LIN {X 0,Y 250.853,Z 488.42,A -85,B 0,C 180,E1 -19750.986,E2 -19750.986} C_VEL
LIN {X 0,Y 251.245,Z 485.6,A -85,B 0,C 180,E1 -19751.504,E2 -19751.504} C_VEL
LIN {X 0,Y 250.177,Z 476.188,A -85,B 0,C 180,E1 -19753.375,E2 -19753.375} C_VEL
LIN {X 0,Y 248.189,Z 466.179,A -85,B 0,C 180,E1 -19755.22,E2 -19755.22} C_VEL
LIN {X 0,Y 245.226,Z 455.953,A -85,B 0,C 180,E1 -19757.02,E2 -19757.02} C_VEL
LIN {X 0,Y 240.964,Z 445.055,A -85,B 0,C 180,E1 -19758.907,E2 -19758.907} C_VEL
LIN {X 0,Y 237.476,Z 437.757,A -85,B 0,C 180,E1 -19760.172,E2 -19760.172} C_VEL
LIN {X 0,Y 236.049,Z 435.07,A -85,B 0,C 180,E1 -19760.656,E2 -19760.656} C_VEL
LIN {X 0,Y 235.755,Z 433.819,A -85,B 0,C 180,E1 -19760.811,E2 -19760.811} C_VEL
LIN {X 0,Y 235.735,Z 432.062,A -85,B 0,C 180,E1 -19763.605,E2 -19763.605} C_VEL
LIN {X 0,Y 235.472,Z 429.817,A -85,B 0,C 180,E1 -19767.505,E2 -19767.505} C_VEL
LIN {X 0,Y 235.182,Z 427.768,A -85,B 0,C 180,E1 -19771.437,E2 -19771.437} C_VEL
LIN {X 0,Y 235.056,Z 426.651,A -85,B 0,C 180,E1 -19773.762,E2 -19773.762} C_VEL
LIN {X 0,Y 234.975,Z 426.216,A -85,B 0,C 180,E1 -19775.246,E2 -19775.246} C_VEL
LIN {X 0,Y 234.995,Z 426.214,A -85,B 0,C 180,E1 -19778.969,E2 -19778.969} C_VEL
LIN {X 0,Y 235.093,Z 426.196,A -85,B 0,C 180,E1 -19783.06,E2 -19783.06} C_VEL
LIN {X 0,Y 235.142,Z 426.195,A -85,B 0,C 180,E1 -19787.924,E2 -19787.924} C_VEL
LIN {X 0,Y 235.374,Z 426.166,A -85,B 0,C 180,E1 -19791.414,E2 -19791.414} C_VEL
LIN {X 0,Y 235.401,Z 426.162,A -85,B 0,C 180,E1 -19793.142,E2 -19793.142} C_VEL
LIN {X 0,Y 235.593,Z 426.139,A -85,B 0,C 180,E1 -19798.291,E2 -19798.291} C_VEL
LIN {X 0,Y 235.593,Z 426.14,A -85,B 0,C 180,E1 -19801.71,E2 -19801.71} C_VEL
LIN {X 0,Y 235.4,Z 426.156,A -85,B 0,C 180,E1 -19806.859,E2 -19806.859} C_VEL
LIN {X 0,Y 235.236,Z 426.183,A -85,B 0,C 180,E1 -19810.327,E2 -19810.327} C_VEL
LIN {X 0,Y 235.112,Z 426.199,A -85,B 0,C 180,E1 -19815.607,E2 -19815.607} C_VEL
LIN {X 0,Y 235.007,Z 426.214,A -85,B 0,C 180,E1 -19819.206,E2 -19819.206} C_VEL
LIN {X 0,Y 234.959,Z 426.222,A -85,B 0,C 180,E1 -19822.883,E2 -19822.883} C_VEL
LIN {X 0,Y 234.969,Z 426.219,A -85,B 0,C 180,E1 -19826.658,E2 -19826.658} C_VEL
LIN {X 0,Y 234.992,Z 426.424,A -85,B 0,C 180,E1 -19829.853,E2 -19829.853} C_VEL
LIN {X 0,Y 235.419,Z 429.003,A -85,B 0,C 180,E1 -19834.556,E2 -19834.556} C_VEL
LIN {X 0,Y 235.897,Z 431.588,A -85,B 0,C 180,E1 -19838.73,E2 -19838.73} C_VEL
LIN {X 0,Y 236.352,Z 434.709,A -85,B 0,C 180,E1 -19843.151,E2 -19843.151} C_VEL
LIN {X 0,Y 236.828,Z 437.629,A -85,B 0,C 180,E1 -19846.958,E2 -19846.958} C_VEL
LIN {X 0,Y 237.155,Z 440.504,A -85,B 0,C 180,E1 -19850.399,E2 -19850.399} C_VEL
LIN {X 0,Y 237.192,Z 441.841,A -85,B 0,C 180,E1 -19851.906,E2 -19851.906} C_VEL
LIN {X 0,Y 237.306,Z 443.408,A -85,B 0,C 180,E1 -19852.73,E2 -19852.73} C_VEL
LIN {X 0,Y 237.585,Z 446.002,A -85,B 0,C 180,E1 -19853.4,E2 -19853.4} C_VEL
LIN {X 0,Y 238.041,Z 450.995,A -85,B 0,C 180,E1 -19854.165,E2 -19854.165} C_VEL
LIN {X 0,Y 238.686,Z 465.72,A -85,B 0,C 180,E1 -19855.664,E2 -19855.664} C_VEL
LIN {X 0,Y 239.11,Z 468.433,A -85,B 0,C 180,E1 -19856.063,E2 -19856.063} C_VEL
LIN {X 0,Y 241.3,Z 479.581,A -85,B 0,C 180,E1 -19857.932,E2 -19857.932} C_VEL
LIN {X 0,Y 242.552,Z 490.657,A -85,B 0,C 180,E1 -19859.937,E2 -19859.937} C_VEL
LIN {X 0,Y 242.646,Z 501.177,A -85,B 0,C 180,E1 -19862.009,E2 -19862.009} C_VEL
LIN {X 0,Y 242.306,Z 505.014,A -85,B 0,C 180,E1 -19862.818,E2 -19862.818} C_VEL
LIN {X 0,Y 239.128,Z 514.446,A -85,B 0,C 180,E1 -19864.776,E2 -19864.776} C_VEL
LIN {X 0,Y 235.867,Z 523.545,A -85,B 0,C 180,E1 -19867.21,E2 -19867.21} C_VEL
LIN {X 0,Y 233.14,Z 530.894,A -85,B 0,C 180,E1 -19869.716,E2 -19869.716} C_VEL
LIN {X 0,Y 230.801,Z 536.822,A -85,B 0,C 180,E1 -19872.272,E2 -19872.272} C_VEL
LIN {X 0,Y 228.794,Z 541.531,A -85,B 0,C 180,E1 -19874.865,E2 -19874.865} C_VEL
LIN {X 0,Y 227.42,Z 545.155,A -85,B 0,C 180,E1 -19877.507,E2 -19877.507} C_VEL
LIN {X 0,Y 226.704,Z 547.044,A -85,B 0,C 180,E1 -19879.28,E2 -19879.28} C_VEL
LIN {X 0,Y 225.834,Z 549.522,A -85,B 0,C 180,E1 -19882.849,E2 -19882.849} C_VEL
LIN {X 0,Y 225.597,Z 550.455,A -85,B 0,C 180,E1 -19886.428,E2 -19886.428} C_VEL
LIN {X 0,Y 225.664,Z 550.323,A -85,B 0,C 180,E1 -19888.215,E2 -19888.215} C_VEL
LIN {X 0,Y 225.758,Z 549.776,A -85,B 0,C 180,E1 -19890,E2 -19890} C_VEL
LIN {X 0,Y 225.69,Z 548.83,A -85,B 0,C 180,E1 -19891.784,E2 -19891.784} C_VEL
LIN {X 0,Y 225.67,Z 546.343,A -85,B 0,C 180,E1 -19894.743,E2 -19894.743} C_VEL
LIN {X 0,Y 225.956,Z 542.13,A -85,B 0,C 180,E1 -19898.045,E2 -19898.045} C_VEL
LIN {X 0,Y 226.522,Z 537.447,A -85,B 0,C 180,E1 -19900.728,E2 -19900.728} C_VEL
LIN {X 0,Y 227.568,Z 530.357,A -85,B 0,C 180,E1 -19903.847,E2 -19903.847} C_VEL
LIN {X 0,Y 229.062,Z 522.678,A -85,B 0,C 180,E1 -19906.487,E2 -19906.487} C_VEL
LIN {X 0,Y 230.612,Z 514.353,A -85,B 0,C 180,E1 -19908.773,E2 -19908.773} C_VEL
LIN {X 0,Y 232.453,Z 504.046,A -85,B 0,C 180,E1 -19911.04,E2 -19911.04} C_VEL
LIN {X 0,Y 233.96,Z 494.379,A -85,B 0,C 180,E1 -19912.752,E2 -19912.752} C_VEL
LIN {X 0,Y 233.445,Z 483.574,A -85,B 0,C 180,E1 -19914.452,E2 -19914.452} C_VEL
LIN {X 0,Y 232.439,Z 471.5,A -85,B 0,C 180,E1 -19915.995,E2 -19915.995} C_VEL
LIN {X 0,Y 230.575,Z 458.277,A -85,B 0,C 180,E1 -19917.362,E2 -19917.362} C_VEL
LIN {X 0,Y 227.792,Z 445.678,A -85,B 0,C 180,E1 -19918.423,E2 -19918.423} C_VEL
LIN {X 0,Y 227.578,Z 444.108,A -85,B 0,C 180,E1 -19918.517,E2 -19918.517} C_VEL
LIN {X 0,Y 228.74,Z 438.72,A -85,B 0,C 180,E1 -19923.575,E2 -19923.575} C_VEL
LIN {X 0,Y 229.126,Z 436.565,A -85,B 0,C 180,E1 -19925.646,E2 -19925.646} C_VEL
LIN {X 0,Y 229.232,Z 434.369,A -85,B 0,C 180,E1 -19927.818,E2 -19927.818} C_VEL
LIN {X 0,Y 228.704,Z 431.101,A -85,B 0,C 180,E1 -19931.273,E2 -19931.273} C_VEL
LIN {X 0,Y 227.914,Z 427.097,A -85,B 0,C 180,E1 -19935.8,E2 -19935.8} C_VEL
LIN {X 0,Y 227.851,Z 427.105,A -85,B 0,C 180,E1 -19940.452,E2 -19940.452} C_VEL
LIN {X 0,Y 227.877,Z 427.099,A -85,B 0,C 180,E1 -19944.127,E2 -19944.127} C_VEL
LIN {X 0,Y 227.867,Z 427.1,A -85,B 0,C 180,E1 -19948.377,E2 -19948.377} C_VEL
LIN {X 0,Y 227.881,Z 427.085,A -85,B 0,C 180,E1 -19952.444,E2 -19952.444} C_VEL
LIN {X 0,Y 227.91,Z 427.094,A -85,B 0,C 180,E1 -19956.367,E2 -19956.367} C_VEL
LIN {X 0,Y 227.936,Z 427.088,A -85,B 0,C 180,E1 -19960.174,E2 -19960.174} C_VEL
LIN {X 0,Y 228.04,Z 427.056,A -85,B 0,C 180,E1 -19963.896,E2 -19963.896} C_VEL
LIN {X 0,Y 228.162,Z 427.062,A -85,B 0,C 180,E1 -19969.349,E2 -19969.349} C_VEL
LIN {X 0,Y 228.354,Z 427.033,A -85,B 0,C 180,E1 -19972.928,E2 -19972.928} C_VEL
LIN {X 0,Y 228.55,Z 426.996,A -85,B 0,C 180,E1 -19978.238,E2 -19978.238} C_VEL
LIN {X 0,Y 228.55,Z 427.011,A -85,B 0,C 180,E1 -19981.762,E2 -19981.762} C_VEL
LIN {X 0,Y 228.35,Z 427.034,A -85,B 0,C 180,E1 -19987.071,E2 -19987.071} C_VEL
LIN {X 0,Y 228.154,Z 427.04,A -85,B 0,C 180,E1 -19990.651,E2 -19990.651} C_VEL
LIN {X 0,Y 228.057,Z 427.067,A -85,B 0,C 180,E1 -19994.272,E2 -19994.272} C_VEL
LIN {X 0,Y 227.998,Z 427.085,A -85,B 0,C 180,E1 -19997.953,E2 -19997.953} C_VEL
LIN {X 0,Y 227.925,Z 427.09,A -85,B 0,C 180,E1 -20002.329,E2 -20002.329} C_VEL
LIN {X 0,Y 227.937,Z 427.09,A -85,B 0,C 180,E1 -20006.603,E2 -20006.603} C_VEL
LIN {X 0,Y 227.893,Z 427.096,A -85,B 0,C 180,E1 -20010.292,E2 -20010.292} C_VEL
LIN {X 0,Y 227.886,Z 427.098,A -85,B 0,C 180,E1 -20013.719,E2 -20013.719} C_VEL
LIN {X 0,Y 227.868,Z 427.1,A -85,B 0,C 180,E1 -20018.086,E2 -20018.086} C_VEL
LIN {X 0,Y 227.93,Z 427.091,A -85,B 0,C 180,E1 -20022.714,E2 -20022.714} C_VEL
LIN {X 0,Y 227.931,Z 427.093,A -85,B 0,C 180,E1 -20027.287,E2 -20027.287} C_VEL
LIN {X 0,Y 227.869,Z 427.1,A -85,B 0,C 180,E1 -20031.915,E2 -20031.915} C_VEL
LIN {X 0,Y 227.888,Z 427.096,A -85,B 0,C 180,E1 -20036.374,E2 -20036.374} C_VEL
LIN {X 0,Y 227.917,Z 427.094,A -85,B 0,C 180,E1 -20040.439,E2 -20040.439} C_VEL
LIN {X 0,Y 227.923,Z 427.093,A -85,B 0,C 180,E1 -20044.426,E2 -20044.426} C_VEL
LIN {X 0,Y 228.038,Z 427.237,A -85,B 0,C 180,E1 -20048.296,E2 -20048.296} C_VEL
LIN {X 0,Y 227.441,Z 431.627,A -85,B 0,C 180,E1 -20053.854,E2 -20053.854} C_VEL
LIN {X 0,Y 227.218,Z 432.967,A -85,B 0,C 180,E1 -20055.503,E2 -20055.503} C_VEL
LIN {X 0,Y 231.479,Z 448.755,A -85,B 0,C 180,E1 -20057.006,E2 -20057.006} C_VEL
LIN {X 0,Y 233.767,Z 459.789,A -85,B 0,C 180,E1 -20058.272,E2 -20058.272} C_VEL
LIN {X 0,Y 235.175,Z 470.256,A -85,B 0,C 180,E1 -20059.671,E2 -20059.671} C_VEL
LIN {X 0,Y 235.635,Z 476.071,A -85,B 0,C 180,E1 -20060.55,E2 -20060.55} C_VEL
LIN {X 0,Y 233.896,Z 487.249,A -85,B 0,C 180,E1 -20062.335,E2 -20062.335} C_VEL
LIN {X 0,Y 232.04,Z 497.341,A -85,B 0,C 180,E1 -20064.351,E2 -20064.351} C_VEL
LIN {X 0,Y 230.343,Z 506,A -85,B 0,C 180,E1 -20066.502,E2 -20066.502} C_VEL
LIN {X 0,Y 228.668,Z 514.397,A -85,B 0,C 180,E1 -20069.12,E2 -20069.12} C_VEL
LIN {X 0,Y 227.487,Z 521.146,A -85,B 0,C 180,E1 -20071.771,E2 -20071.771} C_VEL
LIN {X 0,Y 226.632,Z 526.542,A -85,B 0,C 180,E1 -20074.447,E2 -20074.447} C_VEL
LIN {X 0,Y 226.023,Z 530.762,A -85,B 0,C 180,E1 -20077.145,E2 -20077.145} C_VEL
LIN {X 0,Y 225.696,Z 533.003,A -85,B 0,C 180,E1 -20078.957,E2 -20078.957} C_VEL
LIN {X 0,Y 225.457,Z 534.751,A -85,B 0,C 180,E1 -20080.78,E2 -20080.78} C_VEL
LIN {X 0,Y 225.393,Z 536.082,A -85,B 0,C 180,E1 -20082.607,E2 -20082.607} C_VEL
LIN {X 0,Y 225.404,Z 537.155,A -85,B 0,C 180,E1 -20084.858,E2 -20084.858} C_VEL
LIN {X 0,Y 225.646,Z 537.574,A -85,B 0,C 180,E1 -20088.147,E2 -20088.147} C_VEL
LIN {X 0,Y 226.379,Z 536.717,A -85,B 0,C 180,E1 -20091.353,E2 -20091.353} C_VEL
LIN {X 0,Y 227.101,Z 535.261,A -85,B 0,C 180,E1 -20093.722,E2 -20093.722} C_VEL
LIN {X 0,Y 228.657,Z 532.057,A -85,B 0,C 180,E1 -20096.958,E2 -20096.958} C_VEL
LIN {X 0,Y 230.763,Z 527.351,A -85,B 0,C 180,E1 -20100.166,E2 -20100.166} C_VEL
LIN {X 0,Y 233.107,Z 521.927,A -85,B 0,C 180,E1 -20102.866,E2 -20102.866} C_VEL
LIN {X 0,Y 235.838,Z 515.039,A -85,B 0,C 180,E1 -20105.528,E2 -20105.528} C_VEL
LIN {X 0,Y 238.67,Z 507.605,A -85,B 0,C 180,E1 -20107.787,E2 -20107.787} C_VEL
LIN {X 0,Y 241.524,Z 499.363,A -85,B 0,C 180,E1 -20109.804,E2 -20109.804} C_VEL
LIN {X 0,Y 244.42,Z 490.134,A -85,B 0,C 180,E1 -20111.618,E2 -20111.618} C_VEL
LIN {X 0,Y 244.886,Z 487.509,A -85,B 0,C 180,E1 -20112.103,E2 -20112.103} C_VEL
LIN {X 0,Y 244.042,Z 478.755,A -85,B 0,C 180,E1 -20113.949,E2 -20113.949} C_VEL
LIN {X 0,Y 242.279,Z 468.964,A -85,B 0,C 180,E1 -20115.878,E2 -20115.878} C_VEL
LIN {X 0,Y 239.09,Z 457.518,A -85,B 0,C 180,E1 -20118.031,E2 -20118.031} C_VEL
LIN {X 0,Y 234.687,Z 446.24,A -85,B 0,C 180,E1 -20120.133,E2 -20120.133} C_VEL
LIN {X 0,Y 232.428,Z 441.672,A -85,B 0,C 180,E1 -20121.021,E2 -20121.021} C_VEL
LIN {X 0,Y 230.777,Z 438.365,A -85,B 0,C 180,E1 -20121.648,E2 -20121.648} C_VEL
LIN {X 0,Y 229.134,Z 435.533,A -85,B 0,C 180,E1 -20122.231,E2 -20122.231} C_VEL
LIN {X 0,Y 228.744,Z 434.032,A -85,B 0,C 180,E1 -20122.505,E2 -20122.505} C_VEL
LIN {X 0,Y 228.598,Z 431.802,A -85,B 0,C 180,E1 -20126.4,E2 -20126.4} C_VEL
LIN {X 0,Y 228.31,Z 429.669,A -85,B 0,C 180,E1 -20130.494,E2 -20130.494} C_VEL
LIN {X 0,Y 228.049,Z 427.829,A -85,B 0,C 180,E1 -20134.441,E2 -20134.441} C_VEL
LIN {X 0,Y 227.904,Z 427.095,A -85,B 0,C 180,E1 -20136.367,E2 -20136.367} C_VEL
LIN {X 0,Y 227.934,Z 427.089,A -85,B 0,C 180,E1 -20140.174,E2 -20140.174} C_VEL
LIN {X 0,Y 228.051,Z 427.076,A -85,B 0,C 180,E1 -20143.898,E2 -20143.898} C_VEL
LIN {X 0,Y 228.16,Z 427.058,A -85,B 0,C 180,E1 -20149.35,E2 -20149.35} C_VEL
LIN {X 0,Y 228.352,Z 427.041,A -85,B 0,C 180,E1 -20152.929,E2 -20152.929} C_VEL
LIN {X 0,Y 228.551,Z 427.017,A -85,B 0,C 180,E1 -20158.238,E2 -20158.238} C_VEL
LIN {X 0,Y 228.552,Z 427.017,A -85,B 0,C 180,E1 -20161.762,E2 -20161.762} C_VEL
LIN {X 0,Y 228.351,Z 427.033,A -85,B 0,C 180,E1 -20167.072,E2 -20167.072} C_VEL
LIN {X 0,Y 228.161,Z 427.064,A -85,B 0,C 180,E1 -20170.651,E2 -20170.651} C_VEL
LIN {X 0,Y 228.063,Z 427.077,A -85,B 0,C 180,E1 -20174.273,E2 -20174.273} C_VEL
LIN {X 0,Y 228.001,Z 427.088,A -85,B 0,C 180,E1 -20177.954,E2 -20177.954} C_VEL
LIN {X 0,Y 227.928,Z 427.096,A -85,B 0,C 180,E1 -20182.33,E2 -20182.33} C_VEL
LIN {X 0,Y 227.942,Z 427.094,A -85,B 0,C 180,E1 -20186.603,E2 -20186.603} C_VEL
LIN {X 0,Y 227.885,Z 427.102,A -85,B 0,C 180,E1 -20187.556,E2 -20187.556} C_VEL
LIN {X 0,Y 228.128,Z 428.34,A -85,B 0,C 180,E1 -20190.391,E2 -20190.391} C_VEL
LIN {X 0,Y 228.419,Z 430.171,A -85,B 0,C 180,E1 -20193.827,E2 -20193.827} C_VEL
LIN {X 0,Y 228.828,Z 432.576,A -85,B 0,C 180,E1 -20197.899,E2 -20197.899} C_VEL
LIN {X 0,Y 229.332,Z 435.555,A -85,B 0,C 180,E1 -20202.393,E2 -20202.393} C_VEL
LIN {X 0,Y 229.662,Z 437.646,A -85,B 0,C 180,E1 -20205.265,E2 -20205.265} C_VEL
LIN {X 0,Y 229.943,Z 439.568,A -85,B 0,C 180,E1 -20207.747,E2 -20207.747} C_VEL
LIN {X 0,Y 230.216,Z 442.935,A -85,B 0,C 180,E1 -20211.803,E2 -20211.803} C_VEL
LIN {X 0,Y 230.232,Z 443.288,A -85,B 0,C 180,E1 -20211.988,E2 -20211.988} C_VEL
LIN {X 0,Y 231.387,Z 446.527,A -85,B 0,C 180,E1 -20212.454,E2 -20212.454} C_VEL
LIN {X 0,Y 232.603,Z 448.763,A -85,B 0,C 180,E1 -20212.877,E2 -20212.877} C_VEL
LIN {X 0,Y 236.801,Z 459.979,A -85,B 0,C 180,E1 -20214.704,E2 -20214.704} C_VEL
LIN {X 0,Y 239.11,Z 468.433,A -85,B 0,C 180,E1 -20216.063,E2 -20216.063} C_VEL
LIN {X 0,Y 239.668,Z 473.57,A -85,B 0,C 180,E1 -20216.801,E2 -20216.801} C_VEL
LIN {X 0,Y 238.465,Z 482.57,A -85,B 0,C 180,E1 -20217.875,E2 -20217.875} C_VEL
LIN {X 0,Y 236.768,Z 491.002,A -85,B 0,C 180,E1 -20219.037,E2 -20219.037} C_VEL
LIN {X 0,Y 236.424,Z 495.65,A -85,B 0,C 180,E1 -20219.888,E2 -20219.888} C_VEL
LIN {X 0,Y 235.983,Z 505.59,A -85,B 0,C 180,E1 -20222.027,E2 -20222.027} C_VEL
LIN {X 0,Y 232.755,Z 514.85,A -85,B 0,C 180,E1 -20224.035,E2 -20224.035} C_VEL
LIN {X 0,Y 229.35,Z 523.832,A -85,B 0,C 180,E1 -20226.524,E2 -20226.524} C_VEL
LIN {X 0,Y 226.495,Z 531.095,A -85,B 0,C 180,E1 -20229.094,E2 -20229.094} C_VEL
LIN {X 0,Y 224.042,Z 536.946,A -85,B 0,C 180,E1 -20231.718,E2 -20231.718} C_VEL
LIN {X 0,Y 221.927,Z 541.586,A -85,B 0,C 180,E1 -20234.385,E2 -20234.385} C_VEL
LIN {X 0,Y 220.463,Z 545.144,A -85,B 0,C 180,E1 -20237.106,E2 -20237.106} C_VEL
LIN {X 0,Y 219.709,Z 546.986,A -85,B 0,C 180,E1 -20238.935,E2 -20238.935} C_VEL
LIN {X 0,Y 218.79,Z 549.388,A -85,B 0,C 180,E1 -20242.618,E2 -20242.618} C_VEL
LIN {X 0,Y 218.5,Z 550.258,A -85,B 0,C 180,E1 -20246.311,E2 -20246.311} C_VEL
LIN {X 0,Y 218.579,Z 550.076,A -85,B 0,C 180,E1 -20248.157,E2 -20248.157} C_VEL
LIN {X 0,Y 218.67,Z 549.502,A -85,B 0,C 180,E1 -20250,E2 -20250} C_VEL
LIN {X 0,Y 218.605,Z 548.528,A -85,B 0,C 180,E1 -20251.842,E2 -20251.842} C_VEL
LIN {X 0,Y 218.576,Z 546.262,A -85,B 0,C 180,E1 -20254.609,E2 -20254.609} C_VEL
LIN {X 0,Y 218.78,Z 542.993,A -85,B 0,C 180,E1 -20257.382,E2 -20257.382} C_VEL
LIN {X 0,Y 219.273,Z 538.633,A -85,B 0,C 180,E1 -20260.153,E2 -20260.153} C_VEL
LIN {X 0,Y 220.05,Z 533.053,A -85,B 0,C 180,E1 -20262.918,E2 -20262.918} C_VEL
LIN {X 0,Y 221.421,Z 526.086,A -85,B 0,C 180,E1 -20265.651,E2 -20265.651} C_VEL
LIN {X 0,Y 222.863,Z 518.953,A -85,B 0,C 180,E1 -20267.906,E2 -20267.906} C_VEL
LIN {X 0,Y 224.43,Z 510.287,A -85,B 0,C 180,E1 -20270.148,E2 -20270.148} C_VEL
LIN {X 0,Y 226.435,Z 499.599,A -85,B 0,C 180,E1 -20272.346,E2 -20272.346} C_VEL
LIN {X 0,Y 227.069,Z 494.531,A -85,B 0,C 180,E1 -20273.242,E2 -20273.242} C_VEL
LIN {X 0,Y 226.539,Z 483.294,A -85,B 0,C 180,E1 -20275.074,E2 -20275.074} C_VEL
LIN {X 0,Y 225.552,Z 471.16,A -85,B 0,C 180,E1 -20276.675,E2 -20276.675} C_VEL
LIN {X 0,Y 223.737,Z 458.469,A -85,B 0,C 180,E1 -20278.045,E2 -20278.045} C_VEL
LIN {X 0,Y 220.857,Z 445.431,A -85,B 0,C 180,E1 -20279.199,E2 -20279.199} C_VEL
LIN {X 0,Y 220.63,Z 443.898,A -85,B 0,C 180,E1 -20279.322,E2 -20279.322} C_VEL
LIN {X 0,Y 221.425,Z 440.452,A -85,B 0,C 180,E1 -20282.654,E2 -20282.654} C_VEL
LIN {X 0,Y 222.079,Z 437.223,A -85,B 0,C 180,E1 -20285.834,E2 -20285.834} C_VEL
LIN {X 0,Y 222.202,Z 435.346,A -85,B 0,C 180,E1 -20287.746,E2 -20287.746} C_VEL
LIN {X 0,Y 221.597,Z 431.693,A -85,B 0,C 180,E1 -20291.759,E2 -20291.759} C_VEL
LIN {X 0,Y 220.881,Z 427.973,A -85,B 0,C 180,E1 -20296.196,E2 -20296.196} C_VEL
LIN {X 0,Y 220.805,Z 427.983,A -85,B 0,C 180,E1 -20300.462,E2 -20300.462} C_VEL
LIN {X 0,Y 220.798,Z 427.984,A -85,B 0,C 180,E1 -20305.044,E2 -20305.044} C_VEL
LIN {X 0,Y 220.865,Z 427.969,A -85,B 0,C 180,E1 -20309.394,E2 -20309.394} C_VEL
LIN {X 0,Y 220.891,Z 427.96,A -85,B 0,C 180,E1 -20313.549,E2 -20313.549} C_VEL
LIN {X 0,Y 220.874,Z 427.97,A -85,B 0,C 180,E1 -20317.553,E2 -20317.553} C_VEL
LIN {X 0,Y 220.976,Z 427.938,A -85,B 0,C 180,E1 -20322.574,E2 -20322.574} C_VEL
LIN {X 0,Y 221.003,Z 427.952,A -85,B 0,C 180,E1 -20327.138,E2 -20327.138} C_VEL
LIN {X 0,Y 221.253,Z 427.923,A -85,B 0,C 180,E1 -20330.861,E2 -20330.861} C_VEL
LIN {X 0,Y 221.307,Z 427.911,A -85,B 0,C 180,E1 -20332.702,E2 -20332.702} C_VEL
LIN {X 0,Y 221.508,Z 427.871,A -85,B 0,C 180,E1 -20338.181,E2 -20338.181} C_VEL
LIN {X 0,Y 221.508,Z 427.889,A -85,B 0,C 180,E1 -20341.818,E2 -20341.818} C_VEL
LIN {X 0,Y 221.301,Z 427.912,A -85,B 0,C 180,E1 -20347.298,E2 -20347.298} C_VEL
LIN {X 0,Y 221.101,Z 427.916,A -85,B 0,C 180,E1 -20350.994,E2 -20350.994} C_VEL
LIN {X 0,Y 221.011,Z 427.953,A -85,B 0,C 180,E1 -20356.63,E2 -20356.63} C_VEL
LIN {X 0,Y 220.887,Z 427.966,A -85,B 0,C 180,E1 -20360.486,E2 -20360.486} C_VEL
LIN {X 0,Y 220.862,Z 427.973,A -85,B 0,C 180,E1 -20364.435,E2 -20364.435} C_VEL
LIN {X 0,Y 220.823,Z 427.971,A -85,B 0,C 180,E1 -20368.515,E2 -20368.515} C_VEL
LIN {X 0,Y 220.819,Z 427.977,A -85,B 0,C 180,E1 -20372.755,E2 -20372.755} C_VEL
LIN {X 0,Y 220.834,Z 427.974,A -85,B 0,C 180,E1 -20377.288,E2 -20377.288} C_VEL
LIN {X 0,Y 220.87,Z 427.972,A -85,B 0,C 180,E1 -20381.929,E2 -20381.929} C_VEL
LIN {X 0,Y 220.872,Z 427.973,A -85,B 0,C 180,E1 -20385.573,E2 -20385.573} C_VEL
LIN {X 0,Y 220.858,Z 427.974,A -85,B 0,C 180,E1 -20389.792,E2 -20389.792} C_VEL
LIN {X 0,Y 220.832,Z 427.976,A -85,B 0,C 180,E1 -20392.796,E2 -20392.796} C_VEL
LIN {X 0,Y 220.822,Z 427.979,A -85,B 0,C 180,E1 -20397.246,E2 -20397.246} C_VEL
LIN {X 0,Y 220.835,Z 427.978,A -85,B 0,C 180,E1 -20401.487,E2 -20401.487} C_VEL
LIN {X 0,Y 220.865,Z 427.975,A -85,B 0,C 180,E1 -20405.566,E2 -20405.566} C_VEL
LIN {X 0,Y 220.968,Z 428.041,A -85,B 0,C 180,E1 -20408.056,E2 -20408.056} C_VEL
LIN {X 0,Y 220.428,Z 432.056,A -85,B 0,C 180,E1 -20413.325,E2 -20413.325} C_VEL
LIN {X 0,Y 220.284,Z 433.239,A -85,B 0,C 180,E1 -20414.77,E2 -20414.77} C_VEL
LIN {X 0,Y 223.877,Z 446.278,A -85,B 0,C 180,E1 -20416.004,E2 -20416.004} C_VEL
LIN {X 0,Y 226.646,Z 458.785,A -85,B 0,C 180,E1 -20417.464,E2 -20417.464} C_VEL
LIN {X 0,Y 228.186,Z 469.686,A -85,B 0,C 180,E1 -20418.954,E2 -20418.954} C_VEL
LIN {X 0,Y 228.781,Z 477.32,A -85,B 0,C 180,E1 -20420.151,E2 -20420.151} C_VEL
LIN {X 0,Y 226.956,Z 488.347,A -85,B 0,C 180,E1 -20421.989,E2 -20421.989} C_VEL
LIN {X 0,Y 224.962,Z 498.737,A -85,B 0,C 180,E1 -20424.173,E2 -20424.173} C_VEL
LIN {X 0,Y 223.232,Z 507.152,A -85,B 0,C 180,E1 -20426.39,E2 -20426.39} C_VEL
LIN {X 0,Y 221.521,Z 515.38,A -85,B 0,C 180,E1 -20429.091,E2 -20429.091} C_VEL
LIN {X 0,Y 220.343,Z 521.989,A -85,B 0,C 180,E1 -20431.828,E2 -20431.828} C_VEL
LIN {X 0,Y 219.503,Z 527.258,A -85,B 0,C 180,E1 -20434.591,E2 -20434.591} C_VEL
LIN {X 0,Y 218.866,Z 531.366,A -85,B 0,C 180,E1 -20437.38,E2 -20437.38} C_VEL
LIN {X 0,Y 218.537,Z 533.5,A -85,B 0,C 180,E1 -20439.253,E2 -20439.253} C_VEL
LIN {X 0,Y 218.328,Z 535.192,A -85,B 0,C 180,E1 -20441.136,E2 -20441.136} C_VEL
LIN {X 0,Y 218.274,Z 536.473,A -85,B 0,C 180,E1 -20443.026,E2 -20443.026} C_VEL
LIN {X 0,Y 218.32,Z 537.358,A -85,B 0,C 180,E1 -20445.042,E2 -20445.042} C_VEL
LIN {X 0,Y 218.636,Z 537.758,A -85,B 0,C 180,E1 -20448.75,E2 -20448.75} C_VEL
LIN {X 0,Y 219.372,Z 536.945,A -85,B 0,C 180,E1 -20451.71,E2 -20451.71} C_VEL
LIN {X 0,Y 220.305,Z 535.236,A -85,B 0,C 180,E1 -20454.501,E2 -20454.501} C_VEL
LIN {X 0,Y 221.799,Z 532.335,A -85,B 0,C 180,E1 -20457.475,E2 -20457.475} C_VEL
LIN {X 0,Y 223.595,Z 528.59,A -85,B 0,C 180,E1 -20460.192,E2 -20460.192} C_VEL
LIN {X 0,Y 226.21,Z 522.951,A -85,B 0,C 180,E1 -20463.24,E2 -20463.24} C_VEL
LIN {X 0,Y 229.282,Z 515.724,A -85,B 0,C 180,E1 -20466.161,E2 -20466.161} C_VEL
LIN {X 0,Y 232.646,Z 507.256,A -85,B 0,C 180,E1 -20468.798,E2 -20468.798} C_VEL
LIN {X 0,Y 235.882,Z 498.375,A -85,B 0,C 180,E1 -20470.956,E2 -20470.956} C_VEL
LIN {X 0,Y 238.545,Z 489.774,A -85,B 0,C 180,E1 -20472.658,E2 -20472.658} C_VEL
LIN {X 0,Y 238.001,Z 481.816,A -85,B 0,C 180,E1 -20474.443,E2 -20474.443} C_VEL
LIN {X 0,Y 236.481,Z 472.206,A -85,B 0,C 180,E1 -20476.472,E2 -20476.472} C_VEL
LIN {X 0,Y 233.805,Z 461.655,A -85,B 0,C 180,E1 -20478.601,E2 -20478.601} C_VEL
LIN {X 0,Y 230.13,Z 451.192,A -85,B 0,C 180,E1 -20480.678,E2 -20480.678} C_VEL
LIN {X 0,Y 226.052,Z 442.859,A -85,B 0,C 180,E1 -20482.443,E2 -20482.443} C_VEL
LIN {X 0,Y 223.94,Z 438.84,A -85,B 0,C 180,E1 -20483.299,E2 -20483.299} C_VEL
LIN {X 0,Y 222.162,Z 435.944,A -85,B 0,C 180,E1 -20483.971,E2 -20483.971} C_VEL
LIN {X 0,Y 221.734,Z 434.343,A -85,B 0,C 180,E1 -20484.241,E2 -20484.241} C_VEL
LIN {X 0,Y 221.428,Z 431.852,A -85,B 0,C 180,E1 -20488.976,E2 -20488.976} C_VEL
LIN {X 0,Y 221.184,Z 429.682,A -85,B 0,C 180,E1 -20493.587,E2 -20493.587} C_VEL
LIN {X 0,Y 220.904,Z 428.075,A -85,B 0,C 180,E1 -20497.556,E2 -20497.556} C_VEL
LIN {X 0,Y 220.981,Z 427.955,A -85,B 0,C 180,E1 -20502.572,E2 -20502.572} C_VEL
LIN {X 0,Y 221.021,Z 427.953,A -85,B 0,C 180,E1 -20507.139,E2 -20507.139} C_VEL
LIN {X 0,Y 221.234,Z 427.929,A -85,B 0,C 180,E1 -20510.861,E2 -20510.861} C_VEL
LIN {X 0,Y 221.287,Z 427.922,A -85,B 0,C 180,E1 -20512.702,E2 -20512.702} C_VEL
LIN {X 0,Y 221.51,Z 427.894,A -85,B 0,C 180,E1 -20518.182,E2 -20518.182} C_VEL
LIN {X 0,Y 221.51,Z 427.894,A -85,B 0,C 180,E1 -20521.818,E2 -20521.818} C_VEL
LIN {X 0,Y 221.286,Z 427.912,A -85,B 0,C 180,E1 -20527.299,E2 -20527.299} C_VEL
LIN {X 0,Y 221.11,Z 427.944,A -85,B 0,C 180,E1 -20530.995,E2 -20530.995} C_VEL
LIN {X 0,Y 221.015,Z 427.958,A -85,B 0,C 180,E1 -20536.63,E2 -20536.63} C_VEL
LIN {X 0,Y 220.891,Z 427.973,A -85,B 0,C 180,E1 -20540.487,E2 -20540.487} C_VEL
LIN {X 0,Y 220.866,Z 427.977,A -85,B 0,C 180,E1 -20544.435,E2 -20544.435} C_VEL
LIN {X 0,Y 220.934,Z 428.431,A -85,B 0,C 180,E1 -20547.041,E2 -20547.041} C_VEL
LIN {X 0,Y 221.218,Z 430.234,A -85,B 0,C 180,E1 -20550.933,E2 -20550.933} C_VEL
LIN {X 0,Y 221.569,Z 432.301,A -85,B 0,C 180,E1 -20554.817,E2 -20554.817} C_VEL
LIN {X 0,Y 221.879,Z 433.935,A -85,B 0,C 180,E1 -20557.64,E2 -20557.64} C_VEL
LIN {X 0,Y 222.256,Z 436.44,A -85,B 0,C 180,E1 -20561.61,E2 -20561.61} C_VEL
LIN {X 0,Y 222.791,Z 439.913,A -85,B 0,C 180,E1 -20566.514,E2 -20566.514} C_VEL
LIN {X 0,Y 223.151,Z 442.815,A -85,B 0,C 180,E1 -20570.21,E2 -20570.21} C_VEL
LIN {X 0,Y 224.201,Z 445.876,A -85,B 0,C 180,E1 -20570.682,E2 -20570.682} C_VEL
LIN {X 0,Y 225.802,Z 448.582,A -85,B 0,C 180,E1 -20571.267,E2 -20571.267} C_VEL
LIN {X 0,Y 228.196,Z 454.18,A -85,B 0,C 180,E1 -20572.291,E2 -20572.291} C_VEL
LIN {X 0,Y 231.577,Z 463.952,A -85,B 0,C 180,E1 -20574.026,E2 -20574.026} C_VEL
LIN {X 0,Y 234.295,Z 475.596,A -85,B 0,C 180,E1 -20576.056,E2 -20576.056} C_VEL
LIN {X 0,Y 235.858,Z 486.753,A -85,B 0,C 180,E1 -20578.107,E2 -20578.107} C_VEL
LIN {X 0,Y 236.424,Z 495.65,A -85,B 0,C 180,E1 -20579.888,E2 -20579.888} C_VEL
LIN {X 0,Y 236.097,Z 498.733,A -85,B 0,C 180,E1 -20580.474,E2 -20580.474} C_VEL
LIN {X 0,Y 234.381,Z 503.411,A -85,B 0,C 180,E1 -20581.257,E2 -20581.257} C_VEL
LIN {X 0,Y 231.792,Z 507.929,A -85,B 0,C 180,E1 -20581.98,E2 -20581.98} C_VEL
LIN {X 0,Y 226.978,Z 515.185,A -85,B 0,C 180,E1 -20583.307,E2 -20583.307} C_VEL
LIN {X 0,Y 224.82,Z 519.243,A -85,B 0,C 180,E1 -20584.314,E2 -20584.314} C_VEL
LIN {X 0,Y 221.482,Z 527.49,A -85,B 0,C 180,E1 -20586.959,E2 -20586.959} C_VEL
LIN {X 0,Y 218.942,Z 533.341,A -85,B 0,C 180,E1 -20589.323,E2 -20589.323} C_VEL
LIN {X 0,Y 216.491,Z 538.691,A -85,B 0,C 180,E1 -20592.037,E2 -20592.037} C_VEL
LIN {X 0,Y 214.457,Z 542.891,A -85,B 0,C 180,E1 -20594.801,E2 -20594.801} C_VEL
LIN {X 0,Y 213.525,Z 545.133,A -85,B 0,C 180,E1 -20596.679,E2 -20596.679} C_VEL
LIN {X 0,Y 212.732,Z 546.914,A -85,B 0,C 180,E1 -20598.567,E2 -20598.567} C_VEL
LIN {X 0,Y 211.721,Z 549.256,A -85,B 0,C 180,E1 -20602.37,E2 -20602.37} C_VEL
LIN {X 0,Y 211.421,Z 550.032,A -85,B 0,C 180,E1 -20605.759,E2 -20605.759} C_VEL
LIN {X 0,Y 211.476,Z 549.827,A -85,B 0,C 180,E1 -20608.095,E2 -20608.095} C_VEL
LIN {X 0,Y 211.585,Z 549.224,A -85,B 0,C 180,E1 -20610,E2 -20610} C_VEL
LIN {X 0,Y 211.501,Z 548.22,A -85,B 0,C 180,E1 -20611.904,E2 -20611.904} C_VEL
LIN {X 0,Y 211.474,Z 546.206,A -85,B 0,C 180,E1 -20614.432,E2 -20614.432} C_VEL
LIN {X 0,Y 211.705,Z 542.559,A -85,B 0,C 180,E1 -20617.63,E2 -20617.63} C_VEL
LIN {X 0,Y 212.241,Z 538.131,A -85,B 0,C 180,E1 -20620.493,E2 -20620.493} C_VEL
LIN {X 0,Y 213.085,Z 532.476,A -85,B 0,C 180,E1 -20623.348,E2 -20623.348} C_VEL
LIN {X 0,Y 214.561,Z 525.404,A -85,B 0,C 180,E1 -20626.165,E2 -20626.165} C_VEL
LIN {X 0,Y 216.101,Z 518.172,A -85,B 0,C 180,E1 -20628.486,E2 -20628.486} C_VEL
LIN {X 0,Y 217.492,Z 510.5,A -85,B 0,C 180,E1 -20630.534,E2 -20630.534} C_VEL
LIN {X 0,Y 219.608,Z 499.715,A -85,B 0,C 180,E1 -20632.831,E2 -20632.831} C_VEL
LIN {X 0,Y 220.165,Z 494.66,A -85,B 0,C 180,E1 -20633.765,E2 -20633.765} C_VEL
LIN {X 0,Y 219.744,Z 484.299,A -85,B 0,C 180,E1 -20635.53,E2 -20635.53} C_VEL
LIN {X 0,Y 218.848,Z 472.055,A -85,B 0,C 180,E1 -20637.246,E2 -20637.246} C_VEL
LIN {X 0,Y 217.045,Z 459.375,A -85,B 0,C 180,E1 -20638.699,E2 -20638.699} C_VEL
LIN {X 0,Y 214.261,Z 446.394,A -85,B 0,C 180,E1 -20639.916,E2 -20639.916} C_VEL
LIN {X 0,Y 213.709,Z 443.696,A -85,B 0,C 180,E1 -20640.167,E2 -20640.167} C_VEL
LIN {X 0,Y 214.567,Z 440.038,A -85,B 0,C 180,E1 -20643.835,E2 -20643.835} C_VEL
LIN {X 0,Y 215.127,Z 436.798,A -85,B 0,C 180,E1 -20647.17,E2 -20647.17} C_VEL
LIN {X 0,Y 214.688,Z 433.472,A -85,B 0,C 180,E1 -20650.897,E2 -20650.897} C_VEL
LIN {X 0,Y 214.038,Z 429.921,A -85,B 0,C 180,E1 -20655.094,E2 -20655.094} C_VEL
LIN {X 0,Y 213.819,Z 428.854,A -85,B 0,C 180,E1 -20656.674,E2 -20656.674} C_VEL
LIN {X 0,Y 213.728,Z 428.863,A -85,B 0,C 180,E1 -20662.108,E2 -20662.108} C_VEL
LIN {X 0,Y 213.754,Z 428.858,A -85,B 0,C 180,E1 -20666.017,E2 -20666.017} C_VEL
LIN {X 0,Y 213.777,Z 428.849,A -85,B 0,C 180,E1 -20670.453,E2 -20670.453} C_VEL
LIN {X 0,Y 213.798,Z 428.846,A -85,B 0,C 180,E1 -20674.701,E2 -20674.701} C_VEL
LIN {X 0,Y 213.808,Z 428.85,A -85,B 0,C 180,E1 -20678.803,E2 -20678.803} C_VEL
LIN {X 0,Y 213.934,Z 428.812,A -85,B 0,C 180,E1 -20682.802,E2 -20682.802} C_VEL
LIN {X 0,Y 213.943,Z 428.828,A -85,B 0,C 180,E1 -20686.706,E2 -20686.706} C_VEL
LIN {X 0,Y 214.192,Z 428.805,A -85,B 0,C 180,E1 -20690.557,E2 -20690.557} C_VEL
LIN {X 0,Y 214.243,Z 428.793,A -85,B 0,C 180,E1 -20692.46,E2 -20692.46} C_VEL
LIN {X 0,Y 214.441,Z 428.75,A -85,B 0,C 180,E1 -20698.122,E2 -20698.122} C_VEL
LIN {X 0,Y 214.549,Z 428.748,A -85,B 0,C 180,E1 -20700,E2 -20700} C_VEL
LIN {X 0,Y 214.441,Z 428.769,A -85,B 0,C 180,E1 -20701.878,E2 -20701.878} C_VEL
LIN {X 0,Y 214.235,Z 428.792,A -85,B 0,C 180,E1 -20707.54,E2 -20707.54} C_VEL
LIN {X 0,Y 214.018,Z 428.796,A -85,B 0,C 180,E1 -20711.363,E2 -20711.363} C_VEL
LIN {X 0,Y 213.927,Z 428.829,A -85,B 0,C 180,E1 -20715.237,E2 -20715.237} C_VEL
LIN {X 0,Y 213.835,Z 428.847,A -85,B 0,C 180,E1 -20719.187,E2 -20719.187} C_VEL
LIN {X 0,Y 213.843,Z 428.843,A -85,B 0,C 180,E1 -20723.227,E2 -20723.227} C_VEL
LIN {X 0,Y 213.825,Z 428.849,A -85,B 0,C 180,E1 -20727.45,E2 -20727.45} C_VEL
LIN {X 0,Y 213.766,Z 428.858,A -85,B 0,C 180,E1 -20731.738,E2 -20731.738} C_VEL
LIN {X 0,Y 213.751,Z 428.855,A -85,B 0,C 180,E1 -20736.287,E2 -20736.287} C_VEL
LIN {X 0,Y 213.821,Z 428.849,A -85,B 0,C 180,E1 -20741.099,E2 -20741.099} C_VEL
LIN {X 0,Y 213.833,Z 428.849,A -85,B 0,C 180,E1 -20743.693,E2 -20743.693} C_VEL
LIN {X 0,Y 213.838,Z 428.846,A -85,B 0,C 180,E1 -20746.357,E2 -20746.357} C_VEL
LIN {X 0,Y 213.821,Z 428.85,A -85,B 0,C 180,E1 -20749.11,E2 -20749.11} C_VEL
LIN {X 0,Y 213.752,Z 428.858,A -85,B 0,C 180,E1 -20753.715,E2 -20753.715} C_VEL
LIN {X 0,Y 213.794,Z 428.853,A -85,B 0,C 180,E1 -20758.725,E2 -20758.725} C_VEL
LIN {X 0,Y 213.824,Z 428.85,A -85,B 0,C 180,E1 -20762.604,E2 -20762.604} C_VEL
LIN {X 0,Y 213.938,Z 429.021,A -85,B 0,C 180,E1 -20768.058,E2 -20768.058} C_VEL
LIN {X 0,Y 213.348,Z 433.225,A -85,B 0,C 180,E1 -20773.74,E2 -20773.74} C_VEL
LIN {X 0,Y 213.328,Z 433.365,A -85,B 0,C 180,E1 -20773.923,E2 -20773.923} C_VEL
LIN {X 0,Y 217.107,Z 446.939,A -85,B 0,C 180,E1 -20775.289,E2 -20775.289} C_VEL
LIN {X 0,Y 219.788,Z 459.09,A -85,B 0,C 180,E1 -20776.772,E2 -20776.772} C_VEL
LIN {X 0,Y 221.351,Z 469.972,A -85,B 0,C 180,E1 -20778.323,E2 -20778.323} C_VEL
LIN {X 0,Y 222.003,Z 478.185,A -85,B 0,C 180,E1 -20779.669,E2 -20779.669} C_VEL
LIN {X 0,Y 220.21,Z 488.428,A -85,B 0,C 180,E1 -20781.431,E2 -20781.431} C_VEL
LIN {X 0,Y 218.26,Z 498.231,A -85,B 0,C 180,E1 -20783.529,E2 -20783.529} C_VEL
LIN {X 0,Y 216.442,Z 506.79,A -85,B 0,C 180,E1 -20785.811,E2 -20785.811} C_VEL
LIN {X 0,Y 214.654,Z 515.112,A -85,B 0,C 180,E1 -20788.593,E2 -20788.593} C_VEL
LIN {X 0,Y 213.391,Z 521.807,A -85,B 0,C 180,E1 -20791.416,E2 -20791.416} C_VEL
LIN {X 0,Y 212.353,Z 527.937,A -85,B 0,C 180,E1 -20794.746,E2 -20794.746} C_VEL
LIN {X 0,Y 211.709,Z 531.93,A -85,B 0,C 180,E1 -20797.631,E2 -20797.631} C_VEL
LIN {X 0,Y 211.403,Z 533.989,A -85,B 0,C 180,E1 -20799.568,E2 -20799.568} C_VEL
LIN {X 0,Y 211.199,Z 535.631,A -85,B 0,C 180,E1 -20801.517,E2 -20801.517} C_VEL
LIN {X 0,Y 211.169,Z 536.85,A -85,B 0,C 180,E1 -20803.472,E2 -20803.472} C_VEL
LIN {X 0,Y 211.234,Z 537.613,A -85,B 0,C 180,E1 -20805.436,E2 -20805.436} C_VEL
LIN {X 0,Y 211.376,Z 537.977,A -85,B 0,C 180,E1 -20807.412,E2 -20807.412} C_VEL
LIN {X 0,Y 211.656,Z 537.943,A -85,B 0,C 180,E1 -20809.393,E2 -20809.393} C_VEL
LIN {X 0,Y 212.369,Z 537.174,A -85,B 0,C 180,E1 -20812.088,E2 -20812.088} C_VEL
LIN {X 0,Y 213.537,Z 535.211,A -85,B 0,C 180,E1 -20815.332,E2 -20815.332} C_VEL
LIN {X 0,Y 215,Z 532.586,A -85,B 0,C 180,E1 -20818.045,E2 -20818.045} C_VEL
LIN {X 0,Y 217.149,Z 528.335,A -85,B 0,C 180,E1 -20821.187,E2 -20821.187} C_VEL
LIN {X 0,Y 219.819,Z 522.89,A -85,B 0,C 180,E1 -20824.142,E2 -20824.142} C_VEL
LIN {X 0,Y 222.73,Z 516.413,A -85,B 0,C 180,E1 -20826.835,E2 -20826.835} C_VEL
LIN {X 0,Y 226.155,Z 508.313,A -85,B 0,C 180,E1 -20829.457,E2 -20829.457} C_VEL
LIN {X 0,Y 229.618,Z 499.341,A -85,B 0,C 180,E1 -20831.736,E2 -20831.736} C_VEL
LIN {X 0,Y 232.23,Z 491.21,A -85,B 0,C 180,E1 -20833.422,E2 -20833.422} C_VEL
LIN {X 0,Y 231.735,Z 483.303,A -85,B 0,C 180,E1 -20835.299,E2 -20835.299} C_VEL
LIN {X 0,Y 230.469,Z 474.47,A -85,B 0,C 180,E1 -20837.274,E2 -20837.274} C_VEL
LIN {X 0,Y 228.179,Z 464.783,A -85,B 0,C 180,E1 -20839.367,E2 -20839.367} C_VEL
LIN {X 0,Y 225.12,Z 455.435,A -85,B 0,C 180,E1 -20841.364,E2 -20841.364} C_VEL
LIN {X 0,Y 221.21,Z 447.013,A -85,B 0,C 180,E1 -20843.296,E2 -20843.296} C_VEL
LIN {X 0,Y 219.445,Z 443.603,A -85,B 0,C 180,E1 -20844.093,E2 -20844.093} C_VEL
LIN {X 0,Y 217.257,Z 439.512,A -85,B 0,C 180,E1 -20845.058,E2 -20845.058} C_VEL
LIN {X 0,Y 215.303,Z 436.747,A -85,B 0,C 180,E1 -20845.835,E2 -20845.835} C_VEL
LIN {X 0,Y 214.614,Z 434.647,A -85,B 0,C 180,E1 -20846.243,E2 -20846.243} C_VEL
LIN {X 0,Y 214.369,Z 432.54,A -85,B 0,C 180,E1 -20850.543,E2 -20850.543} C_VEL
LIN {X 0,Y 214.117,Z 430.714,A -85,B 0,C 180,E1 -20854.742,E2 -20854.742} C_VEL
LIN {X 0,Y 213.866,Z 429.179,A -85,B 0,C 180,E1 -20858.809,E2 -20858.809} C_VEL
LIN {X 0,Y 213.94,Z 428.831,A -85,B 0,C 180,E1 -20862.804,E2 -20862.804} C_VEL
LIN {X 0,Y 213.957,Z 428.83,A -85,B 0,C 180,E1 -20866.707,E2 -20866.707} C_VEL
LIN {X 0,Y 214.165,Z 428.808,A -85,B 0,C 180,E1 -20870.557,E2 -20870.557} C_VEL
LIN {X 0,Y 214.225,Z 428.802,A -85,B 0,C 180,E1 -20872.46,E2 -20872.46} C_VEL
LIN {X 0,Y 214.443,Z 428.775,A -85,B 0,C 180,E1 -20878.122,E2 -20878.122} C_VEL
LIN {X 0,Y 214.547,Z 428.761,A -85,B 0,C 180,E1 -20880,E2 -20880} C_VEL
LIN {X 0,Y 214.444,Z 428.774,A -85,B 0,C 180,E1 -20881.878,E2 -20881.878} C_VEL
LIN {X 0,Y 214.224,Z 428.791,A -85,B 0,C 180,E1 -20887.541,E2 -20887.541} C_VEL
LIN {X 0,Y 214.043,Z 428.824,A -85,B 0,C 180,E1 -20891.362,E2 -20891.362} C_VEL
LIN {X 0,Y 213.932,Z 428.838,A -85,B 0,C 180,E1 -20895.237,E2 -20895.237} C_VEL
LIN {X 0,Y 213.838,Z 428.851,A -85,B 0,C 180,E1 -20899.188,E2 -20899.188} C_VEL
LIN {X 0,Y 213.846,Z 428.852,A -85,B 0,C 180,E1 -20903.228,E2 -20903.228} C_VEL
LIN {X 0,Y 214.066,Z 430.316,A -85,B 0,C 180,E1 -20907.573,E2 -20907.573} C_VEL
LIN {X 0,Y 214.326,Z 432.189,A -85,B 0,C 180,E1 -20911.646,E2 -20911.646} C_VEL
LIN {X 0,Y 214.749,Z 434.54,A -85,B 0,C 180,E1 -20916.092,E2 -20916.092} C_VEL
LIN {X 0,Y 215.227,Z 437.325,A -85,B 0,C 180,E1 -20920.775,E2 -20920.775} C_VEL
LIN {X 0,Y 215.734,Z 440.706,A -85,B 0,C 180,E1 -20925.783,E2 -20925.783} C_VEL
LIN {X 0,Y 216.024,Z 442.653,A -85,B 0,C 180,E1 -20928.267,E2 -20928.267} C_VEL
LIN {X 0,Y 217.182,Z 445.761,A -85,B 0,C 180,E1 -20928.81,E2 -20928.81} C_VEL
LIN {X 0,Y 218.866,Z 448.223,A -85,B 0,C 180,E1 -20929.457,E2 -20929.457} C_VEL
LIN {X 0,Y 220.848,Z 452.341,A -85,B 0,C 180,E1 -20930.329,E2 -20930.329} C_VEL
LIN {X 0,Y 223.752,Z 459.429,A -85,B 0,C 180,E1 -20931.744,E2 -20931.744} C_VEL
LIN {X 0,Y 226.775,Z 469.735,A -85,B 0,C 180,E1 -20933.685,E2 -20933.685} C_VEL
LIN {X 0,Y 228.746,Z 480.031,A -85,B 0,C 180,E1 -20935.629,E2 -20935.629} C_VEL
LIN {X 0,Y 229.93,Z 491.069,A -85,B 0,C 180,E1 -20937.834,E2 -20937.834} C_VEL
LIN {X 0,Y 230.064,Z 499.826,A -85,B 0,C 180,E1 -20939.722,E2 -20939.722} C_VEL
LIN {X 0,Y 229.655,Z 506.171,A -85,B 0,C 180,E1 -20941.185,E2 -20941.185} C_VEL
LIN {X 0,Y 227.081,Z 513.577,A -85,B 0,C 180,E1 -20942.839,E2 -20942.839} C_VEL
LIN {X 0,Y 224.82,Z 519.243,A -85,B 0,C 180,E1 -20944.314,E2 -20944.314} C_VEL
LIN {X 0,Y 222.714,Z 523.035,A -85,B 0,C 180,E1 -20945.362,E2 -20945.362} C_VEL
LIN {X 0,Y 217.73,Z 528.783,A -85,B 0,C 180,E1 -20947.03,E2 -20947.03} C_VEL
LIN {X 0,Y 212.825,Z 533.844,A -85,B 0,C 180,E1 -20948.875,E2 -20948.875} C_VEL
LIN {X 0,Y 210.882,Z 536.556,A -85,B 0,C 180,E1 -20950.18,E2 -20950.18} C_VEL
LIN {X 0,Y 208.255,Z 541.671,A -85,B 0,C 180,E1 -20953.331,E2 -20953.331} C_VEL
LIN {X 0,Y 206.584,Z 545.112,A -85,B 0,C 180,E1 -20956.223,E2 -20956.223} C_VEL
LIN {X 0,Y 205.114,Z 548.175,A -85,B 0,C 180,E1 -20960.135,E2 -20960.135} C_VEL
LIN {X 0,Y 204.408,Z 549.687,A -85,B 0,C 180,E1 -20964.079,E2 -20964.079} C_VEL
LIN {X 0,Y 204.337,Z 549.827,A -85,B 0,C 180,E1 -20966.055,E2 -20966.055} C_VEL
LIN {X 0,Y 204.377,Z 549.579,A -85,B 0,C 180,E1 -20968.029,E2 -20968.029} C_VEL
LIN {X 0,Y 204.501,Z 548.947,A -85,B 0,C 180,E1 -20970,E2 -20970} C_VEL
LIN {X 0,Y 204.401,Z 547.912,A -85,B 0,C 180,E1 -20971.97,E2 -20971.97} C_VEL
LIN {X 0,Y 204.38,Z 546.129,A -85,B 0,C 180,E1 -20974.265,E2 -20974.265} C_VEL
LIN {X 0,Y 204.652,Z 542.126,A -85,B 0,C 180,E1 -20977.895,E2 -20977.895} C_VEL
LIN {X 0,Y 205.214,Z 537.628,A -85,B 0,C 180,E1 -20980.856,E2 -20980.856} C_VEL
LIN {X 0,Y 206.381,Z 530.783,A -85,B 0,C 180,E1 -20984.293,E2 -20984.293} C_VEL
LIN {X 0,Y 207.964,Z 523.327,A -85,B 0,C 180,E1 -20987.199,E2 -20987.199} C_VEL
LIN {X 0,Y 209.626,Z 515.715,A -85,B 0,C 180,E1 -20989.588,E2 -20989.588} C_VEL
LIN {X 0,Y 211.044,Z 508.437,A -85,B 0,C 180,E1 -20991.488,E2 -20991.488} C_VEL
LIN {X 0,Y 213.006,Z 498.641,A -85,B 0,C 180,E1 -20993.581,E2 -20993.581} C_VEL
LIN {X 0,Y 213.296,Z 493.443,A -85,B 0,C 180,E1 -20994.581,E2 -20994.581} C_VEL
LIN {X 0,Y 212.847,Z 482.41,A -85,B 0,C 180,E1 -20996.483,E2 -20996.483} C_VEL
LIN {X 0,Y 211.8,Z 470.069,A -85,B 0,C 180,E1 -20998.218,E2 -20998.218} C_VEL
LIN {X 0,Y 210.003,Z 457.999,A -85,B 0,C 180,E1 -20999.628,E2 -20999.628} C_VEL
LIN {X 0,Y 206.971,Z 444.713,A -85,B 0,C 180,E1 -21000.922,E2 -21000.922} C_VEL
LIN {X 0,Y 206.829,Z 443.473,A -85,B 0,C 180,E1 -21001.075,E2 -21001.075} C_VEL
LIN {X 0,Y 207.786,Z 439.622,A -85,B 0,C 180,E1 -21005.098,E2 -21005.098} C_VEL
LIN {X 0,Y 208.073,Z 437.454,A -85,B 0,C 180,E1 -21007.442,E2 -21007.442} C_VEL
LIN {X 0,Y 207.81,Z 435.248,A -85,B 0,C 180,E1 -21009.982,E2 -21009.982} C_VEL
LIN {X 0,Y 207.101,Z 431.479,A -85,B 0,C 180,E1 -21014.55,E2 -21014.55} C_VEL
LIN {X 0,Y 206.76,Z 429.733,A -85,B 0,C 180,E1 -21016.851,E2 -21016.851} C_VEL
LIN {X 0,Y 206.677,Z 429.742,A -85,B 0,C 180,E1 -21022.259,E2 -21022.259} C_VEL
LIN {X 0,Y 206.696,Z 429.74,A -85,B 0,C 180,E1 -21027.041,E2 -21027.041} C_VEL
LIN {X 0,Y 206.763,Z 429.713,A -85,B 0,C 180,E1 -21032.096,E2 -21032.096} C_VEL
LIN {X 0,Y 206.782,Z 429.726,A -85,B 0,C 180,E1 -21036.583,E2 -21036.583} C_VEL
LIN {X 0,Y 206.865,Z 429.697,A -85,B 0,C 180,E1 -21042.195,E2 -21042.195} C_VEL
LIN {X 0,Y 206.884,Z 429.704,A -85,B 0,C 180,E1 -21046.243,E2 -21046.243} C_VEL
LIN {X 0,Y 207.128,Z 429.685,A -85,B 0,C 180,E1 -21050.232,E2 -21050.232} C_VEL
LIN {X 0,Y 207.184,Z 429.674,A -85,B 0,C 180,E1 -21052.201,E2 -21052.201} C_VEL
LIN {X 0,Y 207.378,Z 429.628,A -85,B 0,C 180,E1 -21058.058,E2 -21058.058} C_VEL
LIN {X 0,Y 207.514,Z 429.624,A -85,B 0,C 180,E1 -21060,E2 -21060} C_VEL
LIN {X 0,Y 207.083,Z 429.69,A -85,B 0,C 180,E1 -21063.892,E2 -21063.892} C_VEL
LIN {X 0,Y 207.173,Z 429.669,A -85,B 0,C 180,E1 -21067.798,E2 -21067.798} C_VEL
LIN {X 0,Y 206.938,Z 429.677,A -85,B 0,C 180,E1 -21071.757,E2 -21071.757} C_VEL
LIN {X 0,Y 206.861,Z 429.711,A -85,B 0,C 180,E1 -21075.771,E2 -21075.771} C_VEL
LIN {X 0,Y 206.779,Z 429.728,A -85,B 0,C 180,E1 -21079.869,E2 -21079.869} C_VEL
LIN {X 0,Y 206.759,Z 429.73,A -85,B 0,C 180,E1 -21084.072,E2 -21084.072} C_VEL
LIN {X 0,Y 206.732,Z 429.726,A -85,B 0,C 180,E1 -21088.42,E2 -21088.42} C_VEL
LIN {X 0,Y 206.702,Z 429.736,A -85,B 0,C 180,E1 -21092.957,E2 -21092.957} C_VEL
LIN {X 0,Y 206.722,Z 429.734,A -85,B 0,C 180,E1 -21097.73,E2 -21097.73} C_VEL
LIN {X 0,Y 206.746,Z 429.732,A -85,B 0,C 180,E1 -21101.597,E2 -21101.597} C_VEL
LIN {X 0,Y 206.743,Z 429.732,A -85,B 0,C 180,E1 -21105.55,E2 -21105.55} C_VEL
LIN {X 0,Y 206.741,Z 429.733,A -85,B 0,C 180,E1 -21109.769,E2 -21109.769} C_VEL
LIN {X 0,Y 206.729,Z 429.732,A -85,B 0,C 180,E1 -21114.696,E2 -21114.696} C_VEL
LIN {X 0,Y 206.722,Z 429.735,A -85,B 0,C 180,E1 -21119.34,E2 -21119.34} C_VEL
LIN {X 0,Y 206.731,Z 429.734,A -85,B 0,C 180,E1 -21123.773,E2 -21123.773} C_VEL
LIN {X 0,Y 206.842,Z 429.733,A -85,B 0,C 180,E1 -21127.628,E2 -21127.628} C_VEL
LIN {X 0,Y 206.401,Z 433.366,A -85,B 0,C 180,E1 -21132.734,E2 -21132.734} C_VEL
LIN {X 0,Y 206.4,Z 433.828,A -85,B 0,C 180,E1 -21133.058,E2 -21133.058} C_VEL
LIN {X 0,Y 210.123,Z 446.878,A -85,B 0,C 180,E1 -21134.439,E2 -21134.439} C_VEL
LIN {X 0,Y 212.912,Z 459.099,A -85,B 0,C 180,E1 -21136.001,E2 -21136.001} C_VEL
LIN {X 0,Y 214.572,Z 470.635,A -85,B 0,C 180,E1 -21137.709,E2 -21137.709} C_VEL
LIN {X 0,Y 215.217,Z 478.894,A -85,B 0,C 180,E1 -21139.127,E2 -21139.127} C_VEL
LIN {X 0,Y 213.104,Z 490.369,A -85,B 0,C 180,E1 -21141.202,E2 -21141.202} C_VEL
LIN {X 0,Y 211.19,Z 499.577,A -85,B 0,C 180,E1 -21143.312,E2 -21143.312} C_VEL
LIN {X 0,Y 209.338,Z 507.921,A -85,B 0,C 180,E1 -21145.668,E2 -21145.668} C_VEL
LIN {X 0,Y 207.507,Z 516.088,A -85,B 0,C 180,E1 -21148.545,E2 -21148.545} C_VEL
LIN {X 0,Y 206.448,Z 521.626,A -85,B 0,C 180,E1 -21150.976,E2 -21150.976} C_VEL
LIN {X 0,Y 205.446,Z 527.051,A -85,B 0,C 180,E1 -21153.923,E2 -21153.923} C_VEL
LIN {X 0,Y 204.75,Z 531.296,A -85,B 0,C 180,E1 -21156.899,E2 -21156.899} C_VEL
LIN {X 0,Y 204.247,Z 534.481,A -85,B 0,C 180,E1 -21159.907,E2 -21159.907} C_VEL
LIN {X 0,Y 204.086,Z 536.068,A -85,B 0,C 180,E1 -21161.924,E2 -21161.924} C_VEL
LIN {X 0,Y 204.137,Z 537.759,A -85,B 0,C 180,E1 -21165.426,E2 -21165.426} C_VEL
LIN {X 0,Y 204.36,Z 538.214,A -85,B 0,C 180,E1 -21168.03,E2 -21168.03} C_VEL
LIN {X 0,Y 204.722,Z 538.109,A -85,B 0,C 180,E1 -21170.078,E2 -21170.078} C_VEL
LIN {X 0,Y 205.387,Z 537.4,A -85,B 0,C 180,E1 -21172.498,E2 -21172.498} C_VEL
LIN {X 0,Y 206.814,Z 535.185,A -85,B 0,C 180,E1 -21176.217,E2 -21176.217} C_VEL
LIN {X 0,Y 208.198,Z 532.859,A -85,B 0,C 180,E1 -21178.639,E2 -21178.639} C_VEL
LIN {X 0,Y 210.798,Z 528.077,A -85,B 0,C 180,E1 -21182.238,E2 -21182.238} C_VEL
LIN {X 0,Y 214.057,Z 521.643,A -85,B 0,C 180,E1 -21185.645,E2 -21185.645} C_VEL
LIN {X 0,Y 217.345,Z 514.695,A -85,B 0,C 180,E1 -21188.435,E2 -21188.435} C_VEL
LIN {X 0,Y 220.538,Z 507.259,A -85,B 0,C 180,E1 -21190.789,E2 -21190.789} C_VEL
LIN {X 0,Y 224.48,Z 497.323,A -85,B 0,C 180,E1 -21193.224,E2 -21193.224} C_VEL
LIN {X 0,Y 225.906,Z 493.325,A -85,B 0,C 180,E1 -21194.05,E2 -21194.05} C_VEL
LIN {X 0,Y 225.589,Z 485.41,A -85,B 0,C 180,E1 -21196.052,E2 -21196.052} C_VEL
LIN {X 0,Y 224.379,Z 476.09,A -85,B 0,C 180,E1 -21198.272,E2 -21198.272} C_VEL
LIN {X 0,Y 222.083,Z 466.18,A -85,B 0,C 180,E1 -21200.563,E2 -21200.563} C_VEL
LIN {X 0,Y 219.335,Z 457.827,A -85,B 0,C 180,E1 -21202.497,E2 -21202.497} C_VEL
LIN {X 0,Y 214.85,Z 448.079,A -85,B 0,C 180,E1 -21204.928,E2 -21204.928} C_VEL
LIN {X 0,Y 212.811,Z 444.348,A -85,B 0,C 180,E1 -21205.918,E2 -21205.918} C_VEL
LIN {X 0,Y 210.774,Z 440.563,A -85,B 0,C 180,E1 -21206.907,E2 -21206.907} C_VEL
LIN {X 0,Y 208.232,Z 437.022,A -85,B 0,C 180,E1 -21208.013,E2 -21208.013} C_VEL
LIN {X 0,Y 207.548,Z 434.955,A -85,B 0,C 180,E1 -21208.412,E2 -21208.412} C_VEL
LIN {X 0,Y 207.354,Z 433.459,A -85,B 0,C 180,E1 -21211.791,E2 -21211.791} C_VEL
LIN {X 0,Y 207.052,Z 431.602,A -85,B 0,C 180,E1 -21216.413,E2 -21216.413} C_VEL
LIN {X 0,Y 206.87,Z 429.714,A -85,B 0,C 180,E1 -21222.197,E2 -21222.197} C_VEL
LIN {X 0,Y 206.897,Z 429.707,A -85,B 0,C 180,E1 -21226.245,E2 -21226.245} C_VEL
LIN {X 0,Y 207.104,Z 429.684,A -85,B 0,C 180,E1 -21230.231,E2 -21230.231} C_VEL
LIN {X 0,Y 207.166,Z 429.68,A -85,B 0,C 180,E1 -21232.201,E2 -21232.201} C_VEL
LIN {X 0,Y 207.38,Z 429.655,A -85,B 0,C 180,E1 -21238.058,E2 -21238.058} C_VEL
LIN {X 0,Y 207.512,Z 429.638,A -85,B 0,C 180,E1 -21240,E2 -21240} C_VEL
LIN {X 0,Y 207.38,Z 429.654,A -85,B 0,C 180,E1 -21241.942,E2 -21241.942} C_VEL
LIN {X 0,Y 207.165,Z 429.671,A -85,B 0,C 180,E1 -21247.799,E2 -21247.799} C_VEL
LIN {X 0,Y 206.98,Z 429.702,A -85,B 0,C 180,E1 -21251.756,E2 -21251.756} C_VEL
LIN {X 0,Y 206.865,Z 429.718,A -85,B 0,C 180,E1 -21255.771,E2 -21255.771} C_VEL
LIN {X 0,Y 206.782,Z 429.732,A -85,B 0,C 180,E1 -21259.87,E2 -21259.87} C_VEL
LIN {X 0,Y 206.779,Z 429.903,A -85,B 0,C 180,E1 -21261.955,E2 -21261.955} C_VEL
LIN {X 0,Y 207.049,Z 431.411,A -85,B 0,C 180,E1 -21266.185,E2 -21266.185} C_VEL
LIN {X 0,Y 207.314,Z 433.271,A -85,B 0,C 180,E1 -21270.565,E2 -21270.565} C_VEL
LIN {X 0,Y 207.791,Z 435.854,A -85,B 0,C 180,E1 -21275.735,E2 -21275.735} C_VEL
LIN {X 0,Y 208.169,Z 438.227,A -85,B 0,C 180,E1 -21279.901,E2 -21279.901} C_VEL
LIN {X 0,Y 208.665,Z 441.518,A -85,B 0,C 180,E1 -21285.016,E2 -21285.016} C_VEL
LIN {X 0,Y 208.811,Z 442.244,A -85,B 0,C 180,E1 -21286.051,E2 -21286.051} C_VEL
LIN {X 0,Y 209.829,Z 445.133,A -85,B 0,C 180,E1 -21286.586,E2 -21286.586} C_VEL
LIN {X 0,Y 212.055,Z 448.439,A -85,B 0,C 180,E1 -21287.532,E2 -21287.532} C_VEL
LIN {X 0,Y 214.032,Z 452.309,A -85,B 0,C 180,E1 -21288.469,E2 -21288.469} C_VEL
LIN {X 0,Y 217.362,Z 459.772,A -85,B 0,C 180,E1 -21290.167,E2 -21290.167} C_VEL
LIN {X 0,Y 220.135,Z 468.345,A -85,B 0,C 180,E1 -21291.958,E2 -21291.958} C_VEL
LIN {X 0,Y 222.345,Z 478.771,A -85,B 0,C 180,E1 -21294.062,E2 -21294.062} C_VEL
LIN {X 0,Y 223.593,Z 490.003,A -85,B 0,C 180,E1 -21296.407,E2 -21296.407} C_VEL
LIN {X 0,Y 223.845,Z 499.745,A -85,B 0,C 180,E1 -21298.605,E2 -21298.605} C_VEL
LIN {X 0,Y 223.302,Z 506.721,A -85,B 0,C 180,E1 -21300.284,E2 -21300.284} C_VEL
LIN {X 0,Y 222.246,Z 510.506,A -85,B 0,C 180,E1 -21301.168,E2 -21301.168} C_VEL
LIN {X 0,Y 218.362,Z 519.815,A -85,B 0,C 180,E1 -21303.57,E2 -21303.57} C_VEL
LIN {X 0,Y 214.788,Z 528.173,A -85,B 0,C 180,E1 -21306.374,E2 -21306.374} C_VEL
LIN {X 0,Y 212.31,Z 533.517,A -85,B 0,C 180,E1 -21308.646,E2 -21308.646} C_VEL
LIN {X 0,Y 210.882,Z 536.556,A -85,B 0,C 180,E1 -21310.18,E2 -21310.18} C_VEL
LIN {X 0,Y 209,Z 539.103,A -85,B 0,C 180,E1 -21311.544,E2 -21311.544} C_VEL
LIN {X 0,Y 202.549,Z 543.949,A -85,B 0,C 180,E1 -21314.696,E2 -21314.696} C_VEL
LIN {X 0,Y 199.54,Z 545.994,A -85,B 0,C 180,E1 -21316.698,E2 -21316.698} C_VEL
LIN {X 0,Y 198.76,Z 546.795,A -85,B 0,C 180,E1 -21317.784,E2 -21317.784} C_VEL
LIN {X 0,Y 197.617,Z 548.994,A -85,B 0,C 180,E1 -21321.821,E2 -21321.821} C_VEL
LIN {X 0,Y 197.347,Z 549.504,A -85,B 0,C 180,E1 -21323.867,E2 -21323.867} C_VEL
LIN {X 0,Y 197.281,Z 549.33,A -85,B 0,C 180,E1 -21327.958,E2 -21327.958} C_VEL
LIN {X 0,Y 197.419,Z 548.67,A -85,B 0,C 180,E1 -21330,E2 -21330} C_VEL
LIN {X 0,Y 197.305,Z 547.59,A -85,B 0,C 180,E1 -21332.041,E2 -21332.041} C_VEL
LIN {X 0,Y 197.287,Z 546.053,A -85,B 0,C 180,E1 -21334.085,E2 -21334.085} C_VEL
LIN {X 0,Y 197.463,Z 542.946,A -85,B 0,C 180,E1 -21337.155,E2 -21337.155} C_VEL
LIN {X 0,Y 197.967,Z 538.757,A -85,B 0,C 180,E1 -21340.224,E2 -21340.224} C_VEL
LIN {X 0,Y 199.003,Z 532.342,A -85,B 0,C 180,E1 -21343.79,E2 -21343.79} C_VEL
LIN {X 0,Y 200.575,Z 525.35,A -85,B 0,C 180,E1 -21346.802,E2 -21346.802} C_VEL
LIN {X 0,Y 202.228,Z 518.191,A -85,B 0,C 180,E1 -21349.277,E2 -21349.277} C_VEL
LIN {X 0,Y 203.529,Z 511.544,A -85,B 0,C 180,E1 -21351.198,E2 -21351.198} C_VEL
LIN {X 0,Y 205.521,Z 502.239,A -85,B 0,C 180,E1 -21353.423,E2 -21353.423} C_VEL
LIN {X 0,Y 206.464,Z 496.254,A -85,B 0,C 180,E1 -21354.644,E2 -21354.644} C_VEL
LIN {X 0,Y 206.168,Z 485.822,A -85,B 0,C 180,E1 -21356.608,E2 -21356.608} C_VEL
LIN {X 0,Y 205.471,Z 474.279,A -85,B 0,C 180,E1 -21358.408,E2 -21358.408} C_VEL
LIN {X 0,Y 203.919,Z 461.917,A -85,B 0,C 180,E1 -21360.023,E2 -21360.023} C_VEL
LIN {X 0,Y 201.214,Z 449.005,A -85,B 0,C 180,E1 -21361.434,E2 -21361.434} C_VEL
LIN {X 0,Y 199.964,Z 443.311,A -85,B 0,C 180,E1 -21361.964,E2 -21361.964} C_VEL
LIN {X 0,Y 200.935,Z 439.214,A -85,B 0,C 180,E1 -21366.441,E2 -21366.441} C_VEL
LIN {X 0,Y 200.836,Z 436.465,A -85,B 0,C 180,E1 -21369.658,E2 -21369.658} C_VEL
LIN {X 0,Y 200.4,Z 434.109,A -85,B 0,C 180,E1 -21372.568,E2 -21372.568} C_VEL
LIN {X 0,Y 199.703,Z 430.613,A -85,B 0,C 180,E1 -21377.206,E2 -21377.206} C_VEL
LIN {X 0,Y 199.611,Z 430.625,A -85,B 0,C 180,E1 -21380.766,E2 -21380.766} C_VEL
LIN {X 0,Y 199.609,Z 430.62,A -85,B 0,C 180,E1 -21385.712,E2 -21385.712} C_VEL
LIN {X 0,Y 199.69,Z 430.61,A -85,B 0,C 180,E1 -21388.135,E2 -21388.135} C_VEL
LIN {X 0,Y 199.683,Z 430.594,A -85,B 0,C 180,E1 -21392.771,E2 -21392.771} C_VEL
LIN {X 0,Y 199.734,Z 430.605,A -85,B 0,C 180,E1 -21397.228,E2 -21397.228} C_VEL
LIN {X 0,Y 199.792,Z 430.582,A -85,B 0,C 180,E1 -21401.758,E2 -21401.758} C_VEL
LIN {X 0,Y 199.824,Z 430.581,A -85,B 0,C 180,E1 -21405.747,E2 -21405.747} C_VEL
LIN {X 0,Y 200.071,Z 430.562,A -85,B 0,C 180,E1 -21409.884,E2 -21409.884} C_VEL
LIN {X 0,Y 200.128,Z 430.554,A -85,B 0,C 180,E1 -21411.925,E2 -21411.925} C_VEL
LIN {X 0,Y 200.317,Z 430.506,A -85,B 0,C 180,E1 -21417.989,E2 -21417.989} C_VEL
LIN {X 0,Y 200.478,Z 430.499,A -85,B 0,C 180,E1 -21420,E2 -21420} C_VEL
LIN {X 0,Y 200.029,Z 430.569,A -85,B 0,C 180,E1 -21424.029,E2 -21424.029} C_VEL
LIN {X 0,Y 200.115,Z 430.545,A -85,B 0,C 180,E1 -21428.075,E2 -21428.075} C_VEL
LIN {X 0,Y 199.881,Z 430.557,A -85,B 0,C 180,E1 -21432.179,E2 -21432.179} C_VEL
LIN {X 0,Y 199.799,Z 430.595,A -85,B 0,C 180,E1 -21436.344,E2 -21436.344} C_VEL
LIN {X 0,Y 199.695,Z 430.606,A -85,B 0,C 180,E1 -21440.605,E2 -21440.605} C_VEL
LIN {X 0,Y 199.668,Z 430.612,A -85,B 0,C 180,E1 -21444.985,E2 -21444.985} C_VEL
LIN {X 0,Y 199.661,Z 430.607,A -85,B 0,C 180,E1 -21449.524,E2 -21449.524} C_VEL
LIN {X 0,Y 199.654,Z 430.614,A -85,B 0,C 180,E1 -21452.35,E2 -21452.35} C_VEL
LIN {X 0,Y 199.65,Z 430.611,A -85,B 0,C 180,E1 -21456.757,E2 -21456.757} C_VEL
LIN {X 0,Y 199.698,Z 430.61,A -85,B 0,C 180,E1 -21459.307,E2 -21459.307} C_VEL
LIN {X 0,Y 199.687,Z 430.609,A -85,B 0,C 180,E1 -21462.347,E2 -21462.347} C_VEL
LIN {X 0,Y 199.691,Z 430.611,A -85,B 0,C 180,E1 -21465.262,E2 -21465.262} C_VEL
LIN {X 0,Y 199.696,Z 430.609,A -85,B 0,C 180,E1 -21468.036,E2 -21468.036} C_VEL
LIN {X 0,Y 199.7,Z 430.609,A -85,B 0,C 180,E1 -21470.736,E2 -21470.736} C_VEL
LIN {X 0,Y 199.633,Z 430.618,A -85,B 0,C 180,E1 -21475.719,E2 -21475.719} C_VEL
LIN {X 0,Y 199.702,Z 430.608,A -85,B 0,C 180,E1 -21478.138,E2 -21478.138} C_VEL
LIN {X 0,Y 199.685,Z 430.612,A -85,B 0,C 180,E1 -21482.773,E2 -21482.773} C_VEL
LIN {X 0,Y 199.813,Z 430.663,A -85,B 0,C 180,E1 -21487.512,E2 -21487.512} C_VEL
LIN {X 0,Y 199.38,Z 433.78,A -85,B 0,C 180,E1 -21492.028,E2 -21492.028} C_VEL
LIN {X 0,Y 203.651,Z 448.551,A -85,B 0,C 180,E1 -21493.75,E2 -21493.75} C_VEL
LIN {X 0,Y 206.227,Z 460.321,A -85,B 0,C 180,E1 -21495.344,E2 -21495.344} C_VEL
LIN {X 0,Y 207.612,Z 469.642,A -85,B 0,C 180,E1 -21496.793,E2 -21496.793} C_VEL
LIN {X 0,Y 208.423,Z 479.728,A -85,B 0,C 180,E1 -21498.576,E2 -21498.576} C_VEL
LIN {X 0,Y 206.528,Z 489.794,A -85,B 0,C 180,E1 -21500.451,E2 -21500.451} C_VEL
LIN {X 0,Y 204.545,Z 499.076,A -85,B 0,C 180,E1 -21502.598,E2 -21502.598} C_VEL
LIN {X 0,Y 202.577,Z 507.545,A -85,B 0,C 180,E1 -21505.025,E2 -21505.025} C_VEL
LIN {X 0,Y 200.639,Z 515.813,A -85,B 0,C 180,E1 -21507.993,E2 -21507.993} C_VEL
LIN {X 0,Y 199.321,Z 522.451,A -85,B 0,C 180,E1 -21511.011,E2 -21511.011} C_VEL
LIN {X 0,Y 198.317,Z 527.755,A -85,B 0,C 180,E1 -21514.065,E2 -21514.065} C_VEL
LIN {X 0,Y 197.601,Z 531.891,A -85,B 0,C 180,E1 -21517.151,E2 -21517.151} C_VEL
LIN {X 0,Y 197.114,Z 534.968,A -85,B 0,C 180,E1 -21520.269,E2 -21520.269} C_VEL
LIN {X 0,Y 196.989,Z 536.467,A -85,B 0,C 180,E1 -21522.361,E2 -21522.361} C_VEL
LIN {X 0,Y 197.047,Z 537.957,A -85,B 0,C 180,E1 -21525.636,E2 -21525.636} C_VEL
LIN {X 0,Y 197.355,Z 538.445,A -85,B 0,C 180,E1 -21528.693,E2 -21528.693} C_VEL
LIN {X 0,Y 197.792,Z 538.245,A -85,B 0,C 180,E1 -21530.813,E2 -21530.813} C_VEL
LIN {X 0,Y 198.408,Z 537.632,A -85,B 0,C 180,E1 -21532.932,E2 -21532.932} C_VEL
LIN {X 0,Y 199.173,Z 536.61,A -85,B 0,C 180,E1 -21535.051,E2 -21535.051} C_VEL
LIN {X 0,Y 200.165,Z 535.125,A -85,B 0,C 180,E1 -21537.158,E2 -21537.158} C_VEL
LIN {X 0,Y 202.019,Z 532.151,A -85,B 0,C 180,E1 -21540.178,E2 -21540.178} C_VEL
LIN {X 0,Y 204.52,Z 527.776,A -85,B 0,C 180,E1 -21543.354,E2 -21543.354} C_VEL
LIN {X 0,Y 208.033,Z 521.21,A -85,B 0,C 180,E1 -21546.844,E2 -21546.844} C_VEL
LIN {X 0,Y 210.987,Z 515.266,A -85,B 0,C 180,E1 -21549.263,E2 -21549.263} C_VEL
LIN {X 0,Y 214.246,Z 508.067,A -85,B 0,C 180,E1 -21551.626,E2 -21551.626} C_VEL
LIN {X 0,Y 217.952,Z 499.325,A -85,B 0,C 180,E1 -21553.89,E2 -21553.89} C_VEL
LIN {X 0,Y 219.509,Z 495.272,A -85,B 0,C 180,E1 -21554.778,E2 -21554.778} C_VEL
LIN {X 0,Y 219.6,Z 489.891,A -85,B 0,C 180,E1 -21556.206,E2 -21556.206} C_VEL
LIN {X 0,Y 219.048,Z 482.381,A -85,B 0,C 180,E1 -21558.145,E2 -21558.145} C_VEL
LIN {X 0,Y 217.441,Z 473.109,A -85,B 0,C 180,E1 -21560.46,E2 -21560.46} C_VEL
LIN {X 0,Y 214.919,Z 463.717,A -85,B 0,C 180,E1 -21562.774,E2 -21562.774} C_VEL
LIN {X 0,Y 211.625,Z 455.535,A -85,B 0,C 180,E1 -21564.936,E2 -21564.936} C_VEL
LIN {X 0,Y 208.48,Z 449.222,A -85,B 0,C 180,E1 -21566.712,E2 -21566.712} C_VEL
LIN {X 0,Y 206.094,Z 444.914,A -85,B 0,C 180,E1 -21567.983,E2 -21567.983} C_VEL
LIN {X 0,Y 204.182,Z 441.678,A -85,B 0,C 180,E1 -21568.988,E2 -21568.988} C_VEL
LIN {X 0,Y 203.447,Z 440.4,A -85,B 0,C 180,E1 -21569.368,E2 -21569.368} C_VEL
LIN {X 0,Y 201.316,Z 437.77,A -85,B 0,C 180,E1 -21570.383,E2 -21570.383} C_VEL
LIN {X 0,Y 200.416,Z 435.268,A -85,B 0,C 180,E1 -21571.008,E2 -21571.008} C_VEL
LIN {X 0,Y 200.143,Z 433.322,A -85,B 0,C 180,E1 -21575.92,E2 -21575.92} C_VEL
LIN {X 0,Y 199.931,Z 431.439,A -85,B 0,C 180,E1 -21581.639,E2 -21581.639} C_VEL
LIN {X 0,Y 199.835,Z 430.586,A -85,B 0,C 180,E1 -21585.749,E2 -21585.749} C_VEL
LIN {X 0,Y 200.069,Z 430.558,A -85,B 0,C 180,E1 -21589.884,E2 -21589.884} C_VEL
LIN {X 0,Y 200.032,Z 430.568,A -85,B 0,C 180,E1 -21593.95,E2 -21593.95} C_VEL
LIN {X 0,Y 200.319,Z 430.534,A -85,B 0,C 180,E1 -21597.99,E2 -21597.99} C_VEL
LIN {X 0,Y 200.477,Z 430.514,A -85,B 0,C 180,E1 -21600,E2 -21600} C_VEL
LIN {X 0,Y 200.029,Z 430.569,A -85,B 0,C 180,E1 -21604.03,E2 -21604.03} C_VEL
LIN {X 0,Y 200.109,Z 430.55,A -85,B 0,C 180,E1 -21608.076,E2 -21608.076} C_VEL
LIN {X 0,Y 199.912,Z 430.583,A -85,B 0,C 180,E1 -21612.177,E2 -21612.177} C_VEL
LIN {X 0,Y 199.803,Z 430.6,A -85,B 0,C 180,E1 -21616.344,E2 -21616.344} C_VEL
LIN {X 0,Y 199.783,Z 430.602,A -85,B 0,C 180,E1 -21618.458,E2 -21618.458} C_VEL
LIN {X 0,Y 200.028,Z 432.278,A -85,B 0,C 180,E1 -21624.006,E2 -21624.006} C_VEL
LIN {X 0,Y 200.276,Z 434.07,A -85,B 0,C 180,E1 -21628.684,E2 -21628.684} C_VEL
LIN {X 0,Y 200.549,Z 435.887,A -85,B 0,C 180,E1 -21632.75,E2 -21632.75} C_VEL
LIN {X 0,Y 200.909,Z 437.774,A -85,B 0,C 180,E1 -21636.49,E2 -21636.49} C_VEL
LIN {X 0,Y 201.222,Z 439.603,A -85,B 0,C 180,E1 -21639.792,E2 -21639.792} C_VEL
LIN {X 0,Y 201.54,Z 442.054,A -85,B 0,C 180,E1 -21643.532,E2 -21643.532} C_VEL
LIN {X 0,Y 202.673,Z 445.003,A -85,B 0,C 180,E1 -21644.185,E2 -21644.185} C_VEL
LIN {X 0,Y 205.047,Z 448.225,A -85,B 0,C 180,E1 -21645.291,E2 -21645.291} C_VEL
LIN {X 0,Y 206.925,Z 451.991,A -85,B 0,C 180,E1 -21646.286,E2 -21646.286} C_VEL
LIN {X 0,Y 207.95,Z 453.671,A -85,B 0,C 180,E1 -21646.781,E2 -21646.781} C_VEL
LIN {X 0,Y 211.087,Z 460.474,A -85,B 0,C 180,E1 -21648.514,E2 -21648.514} C_VEL
LIN {X 0,Y 213.548,Z 467.019,A -85,B 0,C 180,E1 -21650.086,E2 -21650.086} C_VEL
LIN {X 0,Y 216.049,Z 477.922,A -85,B 0,C 180,E1 -21652.457,E2 -21652.457} C_VEL
LIN {X 0,Y 217.273,Z 488.248,A -85,B 0,C 180,E1 -21654.714,E2 -21654.714} C_VEL
LIN {X 0,Y 217.668,Z 498.347,A -85,B 0,C 180,E1 -21657.086,E2 -21657.086} C_VEL
LIN {X 0,Y 217.256,Z 505.367,A -85,B 0,C 180,E1 -21658.83,E2 -21658.83} C_VEL
LIN {X 0,Y 216.696,Z 509.166,A -85,B 0,C 180,E1 -21659.821,E2 -21659.821} C_VEL
LIN {X 0,Y 213.179,Z 517.679,A -85,B 0,C 180,E1 -21661.98,E2 -21661.98} C_VEL
LIN {X 0,Y 209.364,Z 526.1,A -85,B 0,C 180,E1 -21664.713,E2 -21664.713} C_VEL
LIN {X 0,Y 205.716,Z 533.694,A -85,B 0,C 180,E1 -21667.926,E2 -21667.926} C_VEL
LIN {X 0,Y 203.028,Z 538.888,A -85,B 0,C 180,E1 -21670.801,E2 -21670.801} C_VEL
LIN {X 0,Y 200.752,Z 542.946,A -85,B 0,C 180,E1 -21673.736,E2 -21673.736} C_VEL
LIN {X 0,Y 199.655,Z 545.079,A -85,B 0,C 180,E1 -21675.735,E2 -21675.735} C_VEL
LIN {X 0,Y 198.76,Z 546.795,A -85,B 0,C 180,E1 -21677.784,E2 -21677.784} C_VEL
LIN {X 0,Y 197.525,Z 547.906,A -85,B 0,C 180,E1 -21679.432,E2 -21679.432} C_VEL
LIN {X 0,Y 194.042,Z 549.056,A -85,B 0,C 180,E1 -21682.129,E2 -21682.129} C_VEL
LIN {X 0,Y 191.364,Z 549.435,A -85,B 0,C 180,E1 -21684.357,E2 -21684.357} C_VEL
LIN {X 0,Y 190.245,Z 549.368,A -85,B 0,C 180,E1 -21686.107,E2 -21686.107} C_VEL
LIN {X 0,Y 190.155,Z 549.281,A -85,B 0,C 180,E1 -21686.701,E2 -21686.701} C_VEL
LIN {X 0,Y 190.319,Z 548.389,A -85,B 0,C 180,E1 -21690,E2 -21690} C_VEL
LIN {X 0,Y 190.179,Z 546.033,A -85,B 0,C 180,E1 -21693.817,E2 -21693.817} C_VEL
LIN {X 0,Y 190.418,Z 542.505,A -85,B 0,C 180,E1 -21697.422,E2 -21697.422} C_VEL
LIN {X 0,Y 190.959,Z 538.244,A -85,B 0,C 180,E1 -21700.603,E2 -21700.603} C_VEL
LIN {X 0,Y 192.075,Z 531.75,A -85,B 0,C 180,E1 -21704.298,E2 -21704.298} C_VEL
LIN {X 0,Y 193.749,Z 524.637,A -85,B 0,C 180,E1 -21707.412,E2 -21707.412} C_VEL
LIN {X 0,Y 195.772,Z 515.714,A -85,B 0,C 180,E1 -21710.487,E2 -21710.487} C_VEL
LIN {X 0,Y 197.483,Z 507.875,A -85,B 0,C 180,E1 -21712.672,E2 -21712.672} C_VEL
LIN {X 0,Y 199.589,Z 497.614,A -85,B 0,C 180,E1 -21714.995,E2 -21714.995} C_VEL
LIN {X 0,Y 199.438,Z 487.776,A -85,B 0,C 180,E1 -21716.98,E2 -21716.98} C_VEL
LIN {X 0,Y 198.905,Z 476.46,A -85,B 0,C 180,E1 -21718.883,E2 -21718.883} C_VEL
LIN {X 0,Y 197.532,Z 464.581,A -85,B 0,C 180,E1 -21720.564,E2 -21720.564} C_VEL
LIN {X 0,Y 195.269,Z 452.655,A -85,B 0,C 180,E1 -21722.001,E2 -21722.001} C_VEL
LIN {X 0,Y 193.136,Z 443.115,A -85,B 0,C 180,E1 -21722.966,E2 -21722.966} C_VEL
LIN {X 0,Y 193.736,Z 440.895,A -85,B 0,C 180,E1 -21725.479,E2 -21725.479} C_VEL
LIN {X 0,Y 193.957,Z 438.727,A -85,B 0,C 180,E1 -21728.023,E2 -21728.023} C_VEL
LIN {X 0,Y 193.629,Z 436.506,A -85,B 0,C 180,E1 -21730.792,E2 -21730.792} C_VEL
LIN {X 0,Y 192.863,Z 432.433,A -85,B 0,C 180,E1 -21736.182,E2 -21736.182} C_VEL
LIN {X 0,Y 192.616,Z 431.496,A -85,B 0,C 180,E1 -21737.87,E2 -21737.87} C_VEL
LIN {X 0,Y 192.584,Z 431.498,A -85,B 0,C 180,E1 -21743.401,E2 -21743.401} C_VEL
LIN {X 0,Y 192.605,Z 431.495,A -85,B 0,C 180,E1 -21747.059,E2 -21747.059} C_VEL
LIN {X 0,Y 192.662,Z 431.469,A -85,B 0,C 180,E1 -21751.691,E2 -21751.691} C_VEL
LIN {X 0,Y 192.702,Z 431.479,A -85,B 0,C 180,E1 -21756.348,E2 -21756.348} C_VEL
LIN {X 0,Y 192.728,Z 431.463,A -85,B 0,C 180,E1 -21761.457,E2 -21761.457} C_VEL
LIN {X 0,Y 192.753,Z 431.456,A -85,B 0,C 180,E1 -21765.212,E2 -21765.212} C_VEL
LIN {X 0,Y 193.016,Z 431.441,A -85,B 0,C 180,E1 -21769.51,E2 -21769.51} C_VEL
LIN {X 0,Y 193,Z 431.432,A -85,B 0,C 180,E1 -21773.728,E2 -21773.728} C_VEL
LIN {X 0,Y 193.259,Z 431.383,A -85,B 0,C 180,E1 -21777.916,E2 -21777.916} C_VEL
LIN {X 0,Y 193.441,Z 431.375,A -85,B 0,C 180,E1 -21780,E2 -21780} C_VEL
LIN {X 0,Y 192.975,Z 431.449,A -85,B 0,C 180,E1 -21784.177,E2 -21784.177} C_VEL
LIN {X 0,Y 193.064,Z 431.42,A -85,B 0,C 180,E1 -21788.372,E2 -21788.372} C_VEL
LIN {X 0,Y 192.804,Z 431.44,A -85,B 0,C 180,E1 -21792.633,E2 -21792.633} C_VEL
LIN {X 0,Y 192.753,Z 431.472,A -85,B 0,C 180,E1 -21796.959,E2 -21796.959} C_VEL
LIN {X 0,Y 192.632,Z 431.485,A -85,B 0,C 180,E1 -21801.397,E2 -21801.397} C_VEL
LIN {X 0,Y 192.66,Z 431.487,A -85,B 0,C 180,E1 -21804.225,E2 -21804.225} C_VEL
LIN {X 0,Y 192.64,Z 431.48,A -85,B 0,C 180,E1 -21808.889,E2 -21808.889} C_VEL
LIN {X 0,Y 192.594,Z 431.494,A -85,B 0,C 180,E1 -21813.186,E2 -21813.186} C_VEL
LIN {X 0,Y 192.61,Z 431.492,A -85,B 0,C 180,E1 -21818.338,E2 -21818.338} C_VEL
LIN {X 0,Y 192.625,Z 431.49,A -85,B 0,C 180,E1 -21823.14,E2 -21823.14} C_VEL
LIN {X 0,Y 192.631,Z 431.488,A -85,B 0,C 180,E1 -21826.86,E2 -21826.86} C_VEL
LIN {X 0,Y 192.611,Z 431.492,A -85,B 0,C 180,E1 -21831.664,E2 -21831.664} C_VEL
LIN {X 0,Y 192.599,Z 431.493,A -85,B 0,C 180,E1 -21836.815,E2 -21836.815} C_VEL
LIN {X 0,Y 192.663,Z 431.487,A -85,B 0,C 180,E1 -21841.693,E2 -21841.693} C_VEL
LIN {X 0,Y 192.777,Z 431.66,A -85,B 0,C 180,E1 -21847.494,E2 -21847.494} C_VEL
LIN {X 0,Y 192.4,Z 434.034,A -85,B 0,C 180,E1 -21851.041,E2 -21851.041} C_VEL
LIN {X 0,Y 194.141,Z 439.438,A -85,B 0,C 180,E1 -21851.652,E2 -21851.652} C_VEL
LIN {X 0,Y 197.511,Z 451.572,A -85,B 0,C 180,E1 -21853.196,E2 -21853.196} C_VEL
LIN {X 0,Y 200.038,Z 464.033,A -85,B 0,C 180,E1 -21855.052,E2 -21855.052} C_VEL
LIN {X 0,Y 201.321,Z 474.76,A -85,B 0,C 180,E1 -21856.886,E2 -21856.886} C_VEL
LIN {X 0,Y 201.675,Z 480.24,A -85,B 0,C 180,E1 -21857.932,E2 -21857.932} C_VEL
LIN {X 0,Y 199.752,Z 490.249,A -85,B 0,C 180,E1 -21859.869,E2 -21859.869} C_VEL
LIN {X 0,Y 197.475,Z 500.373,A -85,B 0,C 180,E1 -21862.331,E2 -21862.331} C_VEL
LIN {X 0,Y 195.103,Z 510.151,A -85,B 0,C 180,E1 -21865.352,E2 -21865.352} C_VEL
LIN {X 0,Y 193.225,Z 517.96,A -85,B 0,C 180,E1 -21868.437,E2 -21868.437} C_VEL
LIN {X 0,Y 192.161,Z 523.269,A -85,B 0,C 180,E1 -21871.048,E2 -21871.048} C_VEL
LIN {X 0,Y 191.182,Z 528.434,A -85,B 0,C 180,E1 -21874.217,E2 -21874.217} C_VEL
LIN {X 0,Y 190.455,Z 532.458,A -85,B 0,C 180,E1 -21877.421,E2 -21877.421} C_VEL
LIN {X 0,Y 189.984,Z 535.438,A -85,B 0,C 180,E1 -21880.659,E2 -21880.659} C_VEL
LIN {X 0,Y 189.879,Z 536.851,A -85,B 0,C 180,E1 -21882.831,E2 -21882.831} C_VEL
LIN {X 0,Y 189.955,Z 538.154,A -85,B 0,C 180,E1 -21885.857,E2 -21885.857} C_VEL
LIN {X 0,Y 190.381,Z 538.639,A -85,B 0,C 180,E1 -21889.405,E2 -21889.405} C_VEL
LIN {X 0,Y 191.456,Z 537.859,A -85,B 0,C 180,E1 -21893.408,E2 -21893.408} C_VEL
LIN {X 0,Y 192.449,Z 536.628,A -85,B 0,C 180,E1 -21895.991,E2 -21895.991} C_VEL
LIN {X 0,Y 194.654,Z 533.42,A -85,B 0,C 180,E1 -21899.943,E2 -21899.943} C_VEL
LIN {X 0,Y 197.385,Z 529.075,A -85,B 0,C 180,E1 -21903.496,E2 -21903.496} C_VEL
LIN {X 0,Y 200.409,Z 523.886,A -85,B 0,C 180,E1 -21906.595,E2 -21906.595} C_VEL
LIN {X 0,Y 203.929,Z 517.249,A -85,B 0,C 180,E1 -21909.61,E2 -21909.61} C_VEL
LIN {X 0,Y 207.999,Z 508.888,A -85,B 0,C 180,E1 -21912.513,E2 -21912.513} C_VEL
LIN {X 0,Y 211.857,Z 500.334,A -85,B 0,C 180,E1 -21914.81,E2 -21914.81} C_VEL
LIN {X 0,Y 213.336,Z 496.566,A -85,B 0,C 180,E1 -21915.678,E2 -21915.678} C_VEL
LIN {X 0,Y 213.339,Z 488.518,A -85,B 0,C 180,E1 -21917.945,E2 -21917.945} C_VEL
LIN {X 0,Y 212.489,Z 480.575,A -85,B 0,C 180,E1 -21920.103,E2 -21920.103} C_VEL
LIN {X 0,Y 210.705,Z 471.554,A -85,B 0,C 180,E1 -21922.503,E2 -21922.503} C_VEL
LIN {X 0,Y 208.84,Z 465.072,A -85,B 0,C 180,E1 -21924.242,E2 -21924.242} C_VEL
LIN {X 0,Y 205.245,Z 456.361,A -85,B 0,C 180,E1 -21926.779,E2 -21926.779} C_VEL
LIN {X 0,Y 201.922,Z 449.906,A -85,B 0,C 180,E1 -21928.82,E2 -21928.82} C_VEL
LIN {X 0,Y 199.617,Z 445.878,A -85,B 0,C 180,E1 -21930.178,E2 -21930.178} C_VEL
LIN {X 0,Y 197.37,Z 442.43,A -85,B 0,C 180,E1 -21931.45,E2 -21931.45} C_VEL
LIN {X 0,Y 196.683,Z 440.987,A -85,B 0,C 180,E1 -21931.882,E2 -21931.882} C_VEL
LIN {X 0,Y 194.446,Z 438.399,A -85,B 0,C 180,E1 -21933.069,E2 -21933.069} C_VEL
LIN {X 0,Y 193.292,Z 435.625,A -85,B 0,C 180,E1 -21933.842,E2 -21933.842} C_VEL
LIN {X 0,Y 193.197,Z 434.682,A -85,B 0,C 180,E1 -21936.413,E2 -21936.413} C_VEL
LIN {X 0,Y 193.015,Z 433.188,A -85,B 0,C 180,E1 -21941.208,E2 -21941.208} C_VEL
LIN {X 0,Y 192.871,Z 432.154,A -85,B 0,C 180,E1 -21945.222,E2 -21945.222} C_VEL
LIN {X 0,Y 192.979,Z 431.439,A -85,B 0,C 180,E1 -21949.509,E2 -21949.509} C_VEL
LIN {X 0,Y 193.06,Z 431.436,A -85,B 0,C 180,E1 -21951.628,E2 -21951.628} C_VEL
LIN {X 0,Y 193.261,Z 431.412,A -85,B 0,C 180,E1 -21957.916,E2 -21957.916} C_VEL
LIN {X 0,Y 193.441,Z 431.391,A -85,B 0,C 180,E1 -21960,E2 -21960} C_VEL
LIN {X 0,Y 192.975,Z 431.447,A -85,B 0,C 180,E1 -21964.177,E2 -21964.177} C_VEL
LIN {X 0,Y 193.06,Z 431.43,A -85,B 0,C 180,E1 -21968.373,E2 -21968.373} C_VEL
LIN {X 0,Y 192.851,Z 431.463,A -85,B 0,C 180,E1 -21972.63,E2 -21972.63} C_VEL
LIN {X 0,Y 192.77,Z 431.503,A -85,B 0,C 180,E1 -21974.786,E2 -21974.786} C_VEL
LIN {X 0,Y 192.873,Z 432.511,A -85,B 0,C 180,E1 -21979.145,E2 -21979.145} C_VEL
LIN {X 0,Y 193.143,Z 434.143,A -85,B 0,C 180,E1 -21984.539,E2 -21984.539} C_VEL
LIN {X 0,Y 193.399,Z 435.937,A -85,B 0,C 180,E1 -21989.293,E2 -21989.293} C_VEL
LIN {X 0,Y 193.678,Z 437.775,A -85,B 0,C 180,E1 -21993.427,E2 -21993.427} C_VEL
LIN {X 0,Y 194.063,Z 440.081,A -85,B 0,C 180,E1 -21998,E2 -21998} C_VEL
LIN {X 0,Y 194.296,Z 441.525,A -85,B 0,C 180,E1 -22000.624,E2 -22000.624} C_VEL
LIN {X 0,Y 195.514,Z 444.7,A -85,B 0,C 180,E1 -22001.425,E2 -22001.425} C_VEL
LIN {X 0,Y 197.983,Z 448.035,A -85,B 0,C 180,E1 -22002.724,E2 -22002.724} C_VEL
LIN {X 0,Y 199.854,Z 451.698,A -85,B 0,C 180,E1 -22003.833,E2 -22003.833} C_VEL
LIN {X 0,Y 201.135,Z 453.637,A -85,B 0,C 180,E1 -22004.509,E2 -22004.509} C_VEL
LIN {X 0,Y 204.128,Z 459.82,A -85,B 0,C 180,E1 -22006.305,E2 -22006.305} C_VEL
LIN {X 0,Y 207.508,Z 467.977,A -85,B 0,C 180,E1 -22008.54,E2 -22008.54} C_VEL
LIN {X 0,Y 209.583,Z 476.048,A -85,B 0,C 180,E1 -22010.468,E2 -22010.468} C_VEL
LIN {X 0,Y 211.028,Z 485.892,A -85,B 0,C 180,E1 -22012.768,E2 -22012.768} C_VEL
LIN {X 0,Y 211.554,Z 495.964,A -85,B 0,C 180,E1 -22015.201,E2 -22015.201} C_VEL
LIN {X 0,Y 211.226,Z 504.937,A -85,B 0,C 180,E1 -22017.538,E2 -22017.538} C_VEL
LIN {X 0,Y 210.524,Z 509.709,A -85,B 0,C 180,E1 -22018.84,E2 -22018.84} C_VEL
LIN {X 0,Y 207.691,Z 516.496,A -85,B 0,C 180,E1 -22020.616,E2 -22020.616} C_VEL
LIN {X 0,Y 203.611,Z 525.022,A -85,B 0,C 180,E1 -22023.339,E2 -22023.339} C_VEL
LIN {X 0,Y 199.708,Z 532.866,A -85,B 0,C 180,E1 -22026.678,E2 -22026.678} C_VEL
LIN {X 0,Y 196.336,Z 538.976,A -85,B 0,C 180,E1 -22030.119,E2 -22030.119} C_VEL
LIN {X 0,Y 193.937,Z 542.97,A -85,B 0,C 180,E1 -22033.147,E2 -22033.147} C_VEL
LIN {X 0,Y 191.808,Z 546.706,A -85,B 0,C 180,E1 -22037.3,E2 -22037.3} C_VEL
LIN {X 0,Y 190.565,Z 548.857,A -85,B 0,C 180,E1 -22041.517,E2 -22041.517} C_VEL
LIN {X 0,Y 190.165,Z 549.386,A -85,B 0,C 180,E1 -22045.761,E2 -22045.761} C_VEL
LIN {X 0,Y 190.155,Z 549.281,A -85,B 0,C 180,E1 -22046.701,E2 -22046.701} C_VEL
LIN {X 0,Y 189.471,Z 548.915,A -85,B 0,C 180,E1 -22048.466,E2 -22048.466} C_VEL
LIN {X 0,Y 187.873,Z 548.202,A -85,B 0,C 180,E1 -22050.193,E2 -22050.193} C_VEL
LIN {X 0,Y 184.188,Z 545.951,A -85,B 0,C 180,E1 -22053.653,E2 -22053.653} C_VEL
LIN {X 0,Y 183.225,Z 544.416,A -85,B 0,C 180,E1 -22055.437,E2 -22055.437} C_VEL
LIN {X 0,Y 183.181,Z 543.831,A -85,B 0,C 180,E1 -22056.037,E2 -22056.037} C_VEL
LIN {X 0,Y 183.714,Z 539.32,A -85,B 0,C 180,E1 -22059.912,E2 -22059.912} C_VEL
LIN {X 0,Y 184.748,Z 533.199,A -85,B 0,C 180,E1 -22063.753,E2 -22063.753} C_VEL
LIN {X 0,Y 186.305,Z 526.491,A -85,B 0,C 180,E1 -22066.998,E2 -22066.998} C_VEL
LIN {X 0,Y 188.392,Z 518.153,A -85,B 0,C 180,E1 -22070.184,E2 -22070.184} C_VEL
LIN {X 0,Y 189.754,Z 511.747,A -85,B 0,C 180,E1 -22072.189,E2 -22072.189} C_VEL
LIN {X 0,Y 191.966,Z 502.35,A -85,B 0,C 180,E1 -22074.609,E2 -22074.609} C_VEL
LIN {X 0,Y 192.755,Z 497.676,A -85,B 0,C 180,E1 -22075.655,E2 -22075.655} C_VEL
LIN {X 0,Y 192.636,Z 486.314,A -85,B 0,C 180,E1 -22078.015,E2 -22078.015} C_VEL
LIN {X 0,Y 191.985,Z 474.461,A -85,B 0,C 180,E1 -22080.038,E2 -22080.038} C_VEL
LIN {X 0,Y 190.549,Z 462.821,A -85,B 0,C 180,E1 -22081.721,E2 -22081.721} C_VEL
LIN {X 0,Y 187.948,Z 450.023,A -85,B 0,C 180,E1 -22083.311,E2 -22083.311} C_VEL
LIN {X 0,Y 186.307,Z 442.912,A -85,B 0,C 180,E1 -22084.074,E2 -22084.074} C_VEL
LIN {X 0,Y 186.831,Z 440.455,A -85,B 0,C 180,E1 -22087.003,E2 -22087.003} C_VEL
LIN {X 0,Y 186.708,Z 438.248,A -85,B 0,C 180,E1 -22089.784,E2 -22089.784} C_VEL
LIN {X 0,Y 186.094,Z 435.005,A -85,B 0,C 180,E1 -22094.147,E2 -22094.147} C_VEL
LIN {X 0,Y 185.578,Z 432.373,A -85,B 0,C 180,E1 -22097.951,E2 -22097.951} C_VEL
LIN {X 0,Y 185.505,Z 432.381,A -85,B 0,C 180,E1 -22102.71,E2 -22102.71} C_VEL
LIN {X 0,Y 185.54,Z 432.372,A -85,B 0,C 180,E1 -22107.974,E2 -22107.974} C_VEL
LIN {X 0,Y 185.579,Z 432.356,A -85,B 0,C 180,E1 -22110.575,E2 -22110.575} C_VEL
LIN {X 0,Y 185.585,Z 432.365,A -85,B 0,C 180,E1 -22115.382,E2 -22115.382} C_VEL
LIN {X 0,Y 185.671,Z 432.342,A -85,B 0,C 180,E1 -22121.133,E2 -22121.133} C_VEL
LIN {X 0,Y 185.685,Z 432.329,A -85,B 0,C 180,E1 -22124.636,E2 -22124.636} C_VEL
LIN {X 0,Y 185.935,Z 432.323,A -85,B 0,C 180,E1 -22129.334,E2 -22129.334} C_VEL
LIN {X 0,Y 185.965,Z 432.31,A -85,B 0,C 180,E1 -22133.49,E2 -22133.49} C_VEL
LIN {X 0,Y 186.203,Z 432.26,A -85,B 0,C 180,E1 -22137.837,E2 -22137.837} C_VEL
LIN {X 0,Y 186.405,Z 432.251,A -85,B 0,C 180,E1 -22140,E2 -22140} C_VEL
LIN {X 0,Y 185.923,Z 432.327,A -85,B 0,C 180,E1 -22144.335,E2 -22144.335} C_VEL
LIN {X 0,Y 186.009,Z 432.297,A -85,B 0,C 180,E1 -22148.692,E2 -22148.692} C_VEL
LIN {X 0,Y 185.729,Z 432.325,A -85,B 0,C 180,E1 -22153.123,E2 -22153.123} C_VEL
LIN {X 0,Y 185.685,Z 432.354,A -85,B 0,C 180,E1 -22157.625,E2 -22157.625} C_VEL
LIN {X 0,Y 185.592,Z 432.36,A -85,B 0,C 180,E1 -22162.252,E2 -22162.252} C_VEL
LIN {X 0,Y 185.556,Z 432.369,A -85,B 0,C 180,E1 -22167.033,E2 -22167.033} C_VEL
LIN {X 0,Y 185.574,Z 432.361,A -85,B 0,C 180,E1 -22169.494,E2 -22169.494} C_VEL
LIN {X 0,Y 185.516,Z 432.37,A -85,B 0,C 180,E1 -22174.628,E2 -22174.628} C_VEL
LIN {X 0,Y 185.564,Z 432.366,A -85,B 0,C 180,E1 -22177.314,E2 -22177.314} C_VEL
LIN {X 0,Y 185.58,Z 432.366,A -85,B 0,C 180,E1 -22180.766,E2 -22180.766} C_VEL
LIN {X 0,Y 185.585,Z 432.366,A -85,B 0,C 180,E1 -22186.014,E2 -22186.014} C_VEL
LIN {X 0,Y 185.565,Z 432.37,A -85,B 0,C 180,E1 -22189.922,E2 -22189.922} C_VEL
LIN {X 0,Y 185.573,Z 432.368,A -85,B 0,C 180,E1 -22192.704,E2 -22192.704} C_VEL
LIN {X 0,Y 185.544,Z 432.373,A -85,B 0,C 180,E1 -22197.976,E2 -22197.976} C_VEL
LIN {X 0,Y 185.581,Z 432.368,A -85,B 0,C 180,E1 -22200.577,E2 -22200.577} C_VEL
LIN {X 0,Y 185.685,Z 432.358,A -85,B 0,C 180,E1 -22206.584,E2 -22206.584} C_VEL
LIN {X 0,Y 185.735,Z 432.841,A -85,B 0,C 180,E1 -22207.767,E2 -22207.767} C_VEL
LIN {X 0,Y 185.466,Z 434.244,A -85,B 0,C 180,E1 -22209.916,E2 -22209.916} C_VEL
LIN {X 0,Y 187.097,Z 439.479,A -85,B 0,C 180,E1 -22210.544,E2 -22210.544} C_VEL
LIN {X 0,Y 190.108,Z 449.44,A -85,B 0,C 180,E1 -22211.897,E2 -22211.897} C_VEL
LIN {X 0,Y 192.495,Z 460.274,A -85,B 0,C 180,E1 -22213.515,E2 -22213.515} C_VEL
LIN {X 0,Y 194.178,Z 470.866,A -85,B 0,C 180,E1 -22215.325,E2 -22215.325} C_VEL
LIN {X 0,Y 194.947,Z 481.001,A -85,B 0,C 180,E1 -22217.291,E2 -22217.291} C_VEL
LIN {X 0,Y 192.739,Z 491.788,A -85,B 0,C 180,E1 -22219.496,E2 -22219.496} C_VEL
LIN {X 0,Y 190.411,Z 501.663,A -85,B 0,C 180,E1 -22222.045,E2 -22222.045} C_VEL
LIN {X 0,Y 188.356,Z 509.767,A -85,B 0,C 180,E1 -22224.648,E2 -22224.648} C_VEL
LIN {X 0,Y 186.352,Z 517.717,A -85,B 0,C 180,E1 -22227.839,E2 -22227.839} C_VEL
LIN {X 0,Y 185.004,Z 524.038,A -85,B 0,C 180,E1 -22231.089,E2 -22231.089} C_VEL
LIN {X 0,Y 184.02,Z 529.077,A -85,B 0,C 180,E1 -22234.381,E2 -22234.381} C_VEL
LIN {X 0,Y 183.306,Z 532.993,A -85,B 0,C 180,E1 -22237.712,E2 -22237.712} C_VEL
LIN {X 0,Y 182.842,Z 535.874,A -85,B 0,C 180,E1 -22241.081,E2 -22241.081} C_VEL
LIN {X 0,Y 182.788,Z 537.234,A -85,B 0,C 180,E1 -22243.338,E2 -22243.338} C_VEL
LIN {X 0,Y 182.87,Z 538.352,A -85,B 0,C 180,E1 -22246.098,E2 -22246.098} C_VEL
LIN {X 0,Y 183.417,Z 538.825,A -85,B 0,C 180,E1 -22250.173,E2 -22250.173} C_VEL
LIN {X 0,Y 184.483,Z 538.096,A -85,B 0,C 180,E1 -22253.895,E2 -22253.895} C_VEL
LIN {X 0,Y 185.784,Z 536.612,A -85,B 0,C 180,E1 -22256.997,E2 -22256.997} C_VEL
LIN {X 0,Y 187.915,Z 533.71,A -85,B 0,C 180,E1 -22260.662,E2 -22260.662} C_VEL
LIN {X 0,Y 191.196,Z 528.837,A -85,B 0,C 180,E1 -22264.733,E2 -22264.733} C_VEL
LIN {X 0,Y 195.067,Z 522.452,A -85,B 0,C 180,E1 -22268.425,E2 -22268.425} C_VEL
LIN {X 0,Y 198.973,Z 515.423,A -85,B 0,C 180,E1 -22271.473,E2 -22271.473} C_VEL
LIN {X 0,Y 202.609,Z 508.18,A -85,B 0,C 180,E1 -22273.927,E2 -22273.927} C_VEL
LIN {X 0,Y 207.009,Z 498.471,A -85,B 0,C 180,E1 -22276.479,E2 -22276.479} C_VEL
LIN {X 0,Y 207.312,Z 492.62,A -85,B 0,C 180,E1 -22278.228,E2 -22278.228} C_VEL
LIN {X 0,Y 206.874,Z 485.06,A -85,B 0,C 180,E1 -22280.434,E2 -22280.434} C_VEL
LIN {X 0,Y 205.434,Z 475.981,A -85,B 0,C 180,E1 -22283.035,E2 -22283.035} C_VEL
LIN {X 0,Y 203.468,Z 468.329,A -85,B 0,C 180,E1 -22285.255,E2 -22285.255} C_VEL
LIN {X 0,Y 199.801,Z 459.21,A -85,B 0,C 180,E1 -22288.155,E2 -22288.155} C_VEL
LIN {X 0,Y 195.757,Z 451.298,A -85,B 0,C 180,E1 -22290.936,E2 -22290.936} C_VEL
LIN {X 0,Y 193.521,Z 447.38,A -85,B 0,C 180,E1 -22292.417,E2 -22292.417} C_VEL
LIN {X 0,Y 190.545,Z 442.939,A -85,B 0,C 180,E1 -22294.298,E2 -22294.298} C_VEL
LIN {X 0,Y 189.897,Z 441.543,A -85,B 0,C 180,E1 -22294.771,E2 -22294.771} C_VEL
LIN {X 0,Y 187.379,Z 438.8,A -85,B 0,C 180,E1 -22296.295,E2 -22296.295} C_VEL
LIN {X 0,Y 186.181,Z 435.97,A -85,B 0,C 180,E1 -22297.237,E2 -22297.237} C_VEL
LIN {X 0,Y 186.041,Z 434.49,A -85,B 0,C 180,E1 -22302.41,E2 -22302.41} C_VEL
LIN {X 0,Y 185.967,Z 433.446,A -85,B 0,C 180,E1 -22306.895,E2 -22306.895} C_VEL
LIN {X 0,Y 186.046,Z 432.649,A -85,B 0,C 180,E1 -22311.31,E2 -22311.31} C_VEL
LIN {X 0,Y 186.206,Z 432.291,A -85,B 0,C 180,E1 -22317.837,E2 -22317.837} C_VEL
LIN {X 0,Y 186.405,Z 432.267,A -85,B 0,C 180,E1 -22320,E2 -22320} C_VEL
LIN {X 0,Y 185.923,Z 432.325,A -85,B 0,C 180,E1 -22324.336,E2 -22324.336} C_VEL
LIN {X 0,Y 186.007,Z 432.31,A -85,B 0,C 180,E1 -22328.693,E2 -22328.693} C_VEL
LIN {X 0,Y 185.862,Z 432.943,A -85,B 0,C 180,E1 -22333.114,E2 -22333.114} C_VEL
LIN {X 0,Y 185.956,Z 433.847,A -85,B 0,C 180,E1 -22337.599,E2 -22337.599} C_VEL
LIN {X 0,Y 186.091,Z 435.077,A -85,B 0,C 180,E1 -22342.19,E2 -22342.19} C_VEL
LIN {X 0,Y 186.255,Z 436.006,A -85,B 0,C 180,E1 -22345.098,E2 -22345.098} C_VEL
LIN {X 0,Y 186.485,Z 437.804,A -85,B 0,C 180,E1 -22349.913,E2 -22349.913} C_VEL
LIN {X 0,Y 186.808,Z 439.762,A -85,B 0,C 180,E1 -22354.356,E2 -22354.356} C_VEL
LIN {X 0,Y 187.113,Z 441.337,A -85,B 0,C 180,E1 -22357.307,E2 -22357.307} C_VEL
LIN {X 0,Y 188.228,Z 444.247,A -85,B 0,C 180,E1 -22358.154,E2 -22358.154} C_VEL
LIN {X 0,Y 190.618,Z 447.148,A -85,B 0,C 180,E1 -22359.578,E2 -22359.578} C_VEL
LIN {X 0,Y 193.168,Z 451.918,A -85,B 0,C 180,E1 -22361.258,E2 -22361.258} C_VEL
LIN {X 0,Y 194.379,Z 453.788,A -85,B 0,C 180,E1 -22361.982,E2 -22361.982} C_VEL
LIN {X 0,Y 196.464,Z 457.742,A -85,B 0,C 180,E1 -22363.345,E2 -22363.345} C_VEL
LIN {X 0,Y 199.54,Z 464.23,A -85,B 0,C 180,E1 -22365.426,E2 -22365.426} C_VEL
LIN {X 0,Y 202.528,Z 472.134,A -85,B 0,C 180,E1 -22367.744,E2 -22367.744} C_VEL
LIN {X 0,Y 204.163,Z 479.564,A -85,B 0,C 180,E1 -22369.653,E2 -22369.653} C_VEL
LIN {X 0,Y 205.242,Z 488.751,A -85,B 0,C 180,E1 -22371.96,E2 -22371.96} C_VEL
LIN {X 0,Y 205.453,Z 498.33,A -85,B 0,C 180,E1 -22374.443,E2 -22374.443} C_VEL
LIN {X 0,Y 204.941,Z 506.535,A -85,B 0,C 180,E1 -22376.724,E2 -22376.724} C_VEL
LIN {X 0,Y 203.871,Z 511.96,A -85,B 0,C 180,E1 -22378.284,E2 -22378.284} C_VEL
LIN {X 0,Y 200.04,Z 519.913,A -85,B 0,C 180,E1 -22380.537,E2 -22380.537} C_VEL
LIN {X 0,Y 196.073,Z 527.739,A -85,B 0,C 180,E1 -22383.382,E2 -22383.382} C_VEL
LIN {X 0,Y 192.649,Z 534.021,A -85,B 0,C 180,E1 -22386.341,E2 -22386.341} C_VEL
LIN {X 0,Y 189.672,Z 539.05,A -85,B 0,C 180,E1 -22389.39,E2 -22389.39} C_VEL
LIN {X 0,Y 187.15,Z 542.977,A -85,B 0,C 180,E1 -22392.517,E2 -22392.517} C_VEL
LIN {X 0,Y 184.864,Z 546.639,A -85,B 0,C 180,E1 -22396.814,E2 -22396.814} C_VEL
LIN {X 0,Y 184.094,Z 547.879,A -85,B 0,C 180,E1 -22398.996,E2 -22398.996} C_VEL
LIN {X 0,Y 183.535,Z 548.703,A -85,B 0,C 180,E1 -22401.189,E2 -22401.189} C_VEL
LIN {X 0,Y 183.079,Z 549.166,A -85,B 0,C 180,E1 -22405.596,E2 -22405.596} C_VEL
LIN {X 0,Y 183.101,Z 548.83,A -85,B 0,C 180,E1 -22407.8,E2 -22407.8} C_VEL
LIN {X 0,Y 183.221,Z 548.096,A -85,B 0,C 180,E1 -22410,E2 -22410} C_VEL
LIN {X 0,Y 183.087,Z 545.971,A -85,B 0,C 180,E1 -22413.58,E2 -22413.58} C_VEL
LIN {X 0,Y 183.181,Z 543.831,A -85,B 0,C 180,E1 -22416.037,E2 -22416.037} C_VEL
LIN {X 0,Y 182.672,Z 541.979,A -85,B 0,C 180,E1 -22417.788,E2 -22417.788} C_VEL
LIN {X 0,Y 180.245,Z 538.403,A -85,B 0,C 180,E1 -22420.612,E2 -22420.612} C_VEL
LIN {X 0,Y 178.127,Z 534.14,A -85,B 0,C 180,E1 -22423.411,E2 -22423.411} C_VEL
LIN {X 0,Y 178.116,Z 531.203,A -85,B 0,C 180,E1 -22425.071,E2 -22425.071} C_VEL
LIN {X 0,Y 179.83,Z 524.553,A -85,B 0,C 180,E1 -22428.218,E2 -22428.218} C_VEL
LIN {X 0,Y 181.906,Z 516.136,A -85,B 0,C 180,E1 -22431.373,E2 -22431.373} C_VEL
LIN {X 0,Y 183.611,Z 508.969,A -85,B 0,C 180,E1 -22433.577,E2 -22433.577} C_VEL
LIN {X 0,Y 185.91,Z 498.951,A -85,B 0,C 180,E1 -22436.069,E2 -22436.069} C_VEL
LIN {X 0,Y 185.932,Z 488.228,A -85,B 0,C 180,E1 -22438.45,E2 -22438.45} C_VEL
LIN {X 0,Y 185.472,Z 476.819,A -85,B 0,C 180,E1 -22440.566,E2 -22440.566} C_VEL
LIN {X 0,Y 184.234,Z 465.192,A -85,B 0,C 180,E1 -22442.384,E2 -22442.384} C_VEL
LIN {X 0,Y 181.689,Z 452.039,A -85,B 0,C 180,E1 -22444.161,E2 -22444.161} C_VEL
LIN {X 0,Y 179.509,Z 442.694,A -85,B 0,C 180,E1 -22445.273,E2 -22445.273} C_VEL
LIN {X 0,Y 179.812,Z 441.143,A -85,B 0,C 180,E1 -22447.213,E2 -22447.213} C_VEL
LIN {X 0,Y 179.626,Z 438.874,A -85,B 0,C 180,E1 -22450.207,E2 -22450.207} C_VEL
LIN {X 0,Y 178.964,Z 435.467,A -85,B 0,C 180,E1 -22455.019,E2 -22455.019} C_VEL
LIN {X 0,Y 178.501,Z 433.255,A -85,B 0,C 180,E1 -22458.422,E2 -22458.422} C_VEL
LIN {X 0,Y 178.42,Z 433.261,A -85,B 0,C 180,E1 -22463.782,E2 -22463.782} C_VEL
LIN {X 0,Y 178.483,Z 433.253,A -85,B 0,C 180,E1 -22466.545,E2 -22466.545} C_VEL
LIN {X 0,Y 178.52,Z 433.241,A -85,B 0,C 180,E1 -22470.006,E2 -22470.006} C_VEL
LIN {X 0,Y 178.532,Z 433.238,A -85,B 0,C 180,E1 -22474.875,E2 -22474.875} C_VEL
LIN {X 0,Y 178.619,Z 433.222,A -85,B 0,C 180,E1 -22480.784,E2 -22480.784} C_VEL
LIN {X 0,Y 178.653,Z 433.218,A -85,B 0,C 180,E1 -22486.347,E2 -22486.347} C_VEL
LIN {X 0,Y 178.973,Z 433.189,A -85,B 0,C 180,E1 -22490.963,E2 -22490.963} C_VEL
LIN {X 0,Y 179.149,Z 433.137,A -85,B 0,C 180,E1 -22497.751,E2 -22497.751} C_VEL
LIN {X 0,Y 179.368,Z 433.127,A -85,B 0,C 180,E1 -22500,E2 -22500} C_VEL
LIN {X 0,Y 178.871,Z 433.204,A -85,B 0,C 180,E1 -22504.507,E2 -22504.507} C_VEL
LIN {X 0,Y 178.959,Z 433.171,A -85,B 0,C 180,E1 -22509.037,E2 -22509.037} C_VEL
LIN {X 0,Y 178.656,Z 433.21,A -85,B 0,C 180,E1 -22513.652,E2 -22513.652} C_VEL
LIN {X 0,Y 178.619,Z 433.234,A -85,B 0,C 180,E1 -22519.216,E2 -22519.216} C_VEL
LIN {X 0,Y 178.52,Z 433.247,A -85,B 0,C 180,E1 -22525.118,E2 -22525.118} C_VEL
LIN {X 0,Y 178.518,Z 433.242,A -85,B 0,C 180,E1 -22529.993,E2 -22529.993} C_VEL
LIN {X 0,Y 178.48,Z 433.248,A -85,B 0,C 180,E1 -22534.219,E2 -22534.219} C_VEL
LIN {X 0,Y 178.482,Z 433.252,A -85,B 0,C 180,E1 -22539.051,E2 -22539.051} C_VEL
LIN {X 0,Y 178.511,Z 433.248,A -85,B 0,C 180,E1 -22542.012,E2 -22542.012} C_VEL
LIN {X 0,Y 178.527,Z 433.247,A -85,B 0,C 180,E1 -22545.12,E2 -22545.12} C_VEL
LIN {X 0,Y 178.517,Z 433.247,A -85,B 0,C 180,E1 -22548.418,E2 -22548.418} C_VEL
LIN {X 0,Y 178.466,Z 433.253,A -85,B 0,C 180,E1 -22553.795,E2 -22553.795} C_VEL
LIN {X 0,Y 178.49,Z 433.25,A -85,B 0,C 180,E1 -22556.549,E2 -22556.549} C_VEL
LIN {X 0,Y 178.521,Z 433.248,A -85,B 0,C 180,E1 -22560.007,E2 -22560.007} C_VEL
LIN {X 0,Y 178.655,Z 433.25,A -85,B 0,C 180,E1 -22566.765,E2 -22566.765} C_VEL
LIN {X 0,Y 178.596,Z 434.434,A -85,B 0,C 180,E1 -22568.716,E2 -22568.716} C_VEL
LIN {X 0,Y 180.326,Z 440.041,A -85,B 0,C 180,E1 -22569.422,E2 -22569.422} C_VEL
LIN {X 0,Y 183.472,Z 450.167,A -85,B 0,C 180,E1 -22570.909,E2 -22570.909} C_VEL
LIN {X 0,Y 185.885,Z 461.149,A -85,B 0,C 180,E1 -22572.653,E2 -22572.653} C_VEL
LIN {X 0,Y 187.624,Z 472.957,A -85,B 0,C 180,E1 -22574.8,E2 -22574.8} C_VEL
LIN {X 0,Y 188.223,Z 481.986,A -85,B 0,C 180,E1 -22576.657,E2 -22576.657} C_VEL
LIN {X 0,Y 186.211,Z 491.436,A -85,B 0,C 180,E1 -22578.653,E2 -22578.653} C_VEL
LIN {X 0,Y 183.804,Z 501.148,A -85,B 0,C 180,E1 -22581.203,E2 -22581.203} C_VEL
LIN {X 0,Y 181.254,Z 510.866,A -85,B 0,C 180,E1 -22584.438,E2 -22584.438} C_VEL
LIN {X 0,Y 179.227,Z 518.599,A -85,B 0,C 180,E1 -22587.753,E2 -22587.753} C_VEL
LIN {X 0,Y 177.852,Z 524.79,A -85,B 0,C 180,E1 -22591.133,E2 -22591.133} C_VEL
LIN {X 0,Y 176.867,Z 529.715,A -85,B 0,C 180,E1 -22594.559,E2 -22594.559} C_VEL
LIN {X 0,Y 176.138,Z 533.526,A -85,B 0,C 180,E1 -22598.028,E2 -22598.028} C_VEL
LIN {X 0,Y 175.709,Z 536.305,A -85,B 0,C 180,E1 -22601.537,E2 -22601.537} C_VEL
LIN {X 0,Y 175.678,Z 537.616,A -85,B 0,C 180,E1 -22603.888,E2 -22603.888} C_VEL
LIN {X 0,Y 175.799,Z 538.55,A -85,B 0,C 180,E1 -22606.371,E2 -22606.371} C_VEL
LIN {X 0,Y 176.046,Z 538.967,A -85,B 0,C 180,E1 -22608.625,E2 -22608.625} C_VEL
LIN {X 0,Y 176.484,Z 539.012,A -85,B 0,C 180,E1 -22611.002,E2 -22611.002} C_VEL
LIN {X 0,Y 177.537,Z 538.333,A -85,B 0,C 180,E1 -22614.429,E2 -22614.429} C_VEL
LIN {X 0,Y 179.162,Z 536.598,A -85,B 0,C 180,E1 -22618.081,E2 -22618.081} C_VEL
LIN {X 0,Y 181.226,Z 533.993,A -85,B 0,C 180,E1 -22621.443,E2 -22621.443} C_VEL
LIN {X 0,Y 184.055,Z 530.076,A -85,B 0,C 180,E1 -22624.943,E2 -22624.943} C_VEL
LIN {X 0,Y 187.551,Z 524.79,A -85,B 0,C 180,E1 -22628.382,E2 -22628.382} C_VEL
LIN {X 0,Y 191.259,Z 518.65,A -85,B 0,C 180,E1 -22631.408,E2 -22631.408} C_VEL
LIN {X 0,Y 195.646,Z 510.69,A -85,B 0,C 180,E1 -22634.398,E2 -22634.398} C_VEL
LIN {X 0,Y 199.864,Z 502.2,A -85,B 0,C 180,E1 -22636.856,E2 -22636.856} C_VEL
LIN {X 0,Y 201.088,Z 498.852,A -85,B 0,C 180,E1 -22637.757,E2 -22637.757} C_VEL
LIN {X 0,Y 201.139,Z 489.916,A -85,B 0,C 180,E1 -22640.608,E2 -22640.608} C_VEL
LIN {X 0,Y 200.19,Z 480.977,A -85,B 0,C 180,E1 -22643.358,E2 -22643.358} C_VEL
LIN {X 0,Y 198.742,Z 473.92,A -85,B 0,C 180,E1 -22645.543,E2 -22645.543} C_VEL
LIN {X 0,Y 195.627,Z 464.796,A -85,B 0,C 180,E1 -22648.606,E2 -22648.606} C_VEL
LIN {X 0,Y 191.915,Z 456.893,A -85,B 0,C 180,E1 -22651.572,E2 -22651.572} C_VEL
LIN {X 0,Y 188.377,Z 450.883,A -85,B 0,C 180,E1 -22654.149,E2 -22654.149} C_VEL
LIN {X 0,Y 186.446,Z 447.293,A -85,B 0,C 180,E1 -22655.652,E2 -22655.652} C_VEL
LIN {X 0,Y 184.145,Z 444.277,A -85,B 0,C 180,E1 -22657.268,E2 -22657.268} C_VEL
LIN {X 0,Y 183.079,Z 442.092,A -85,B 0,C 180,E1 -22658.169,E2 -22658.169} C_VEL
LIN {X 0,Y 180.715,Z 439.856,A -85,B 0,C 180,E1 -22659.842,E2 -22659.842} C_VEL
LIN {X 0,Y 179.326,Z 437.004,A -85,B 0,C 180,E1 -22661.103,E2 -22661.103} C_VEL
LIN {X 0,Y 179.151,Z 436.399,A -85,B 0,C 180,E1 -22661.334,E2 -22661.334} C_VEL
LIN {X 0,Y 179.044,Z 435.224,A -85,B 0,C 180,E1 -22666.378,E2 -22666.378} C_VEL
LIN {X 0,Y 179.138,Z 434.397,A -85,B 0,C 180,E1 -22670.972,E2 -22670.972} C_VEL
LIN {X 0,Y 179.238,Z 433.733,A -85,B 0,C 180,E1 -22677.753,E2 -22677.753} C_VEL
LIN {X 0,Y 179.447,Z 433.604,A -85,B 0,C 180,E1 -22680,E2 -22680} C_VEL
LIN {X 0,Y 179.056,Z 433.89,A -85,B 0,C 180,E1 -22686.763,E2 -22686.763} C_VEL
LIN {X 0,Y 179.12,Z 434.089,A -85,B 0,C 180,E1 -22689.03,E2 -22689.03} C_VEL
LIN {X 0,Y 178.962,Z 434.793,A -85,B 0,C 180,E1 -22693.629,E2 -22693.629} C_VEL
LIN {X 0,Y 179.074,Z 435.736,A -85,B 0,C 180,E1 -22698.299,E2 -22698.299} C_VEL
LIN {X 0,Y 179.223,Z 437.044,A -85,B 0,C 180,E1 -22703.088,E2 -22703.088} C_VEL
LIN {X 0,Y 179.469,Z 438.688,A -85,B 0,C 180,E1 -22708.03,E2 -22708.03} C_VEL
LIN {X 0,Y 179.796,Z 440.848,A -85,B 0,C 180,E1 -22713.178,E2 -22713.178} C_VEL
LIN {X 0,Y 180.908,Z 443.649,A -85,B 0,C 180,E1 -22714.199,E2 -22714.199} C_VEL
LIN {X 0,Y 183.126,Z 446.545,A -85,B 0,C 180,E1 -22715.823,E2 -22715.823} C_VEL
LIN {X 0,Y 184.045,Z 447.533,A -85,B 0,C 180,E1 -22716.433,E2 -22716.433} C_VEL
LIN {X 0,Y 185.9,Z 451.309,A -85,B 0,C 180,E1 -22717.906,E2 -22717.906} C_VEL
LIN {X 0,Y 187.654,Z 453.713,A -85,B 0,C 180,E1 -22719.077,E2 -22719.077} C_VEL
LIN {X 0,Y 189.763,Z 457.845,A -85,B 0,C 180,E1 -22720.663,E2 -22720.663} C_VEL
LIN {X 0,Y 190.259,Z 458.48,A -85,B 0,C 180,E1 -22720.971,E2 -22720.971} C_VEL
LIN {X 0,Y 194.69,Z 468.047,A -85,B 0,C 180,E1 -22724.374,E2 -22724.374} C_VEL
LIN {X 0,Y 197.421,Z 476.011,A -85,B 0,C 180,E1 -22726.87,E2 -22726.87} C_VEL
LIN {X 0,Y 198.827,Z 483.808,A -85,B 0,C 180,E1 -22729.03,E2 -22729.03} C_VEL
LIN {X 0,Y 199.506,Z 493.622,A -85,B 0,C 180,E1 -22731.677,E2 -22731.677} C_VEL
LIN {X 0,Y 199.208,Z 503.349,A -85,B 0,C 180,E1 -22734.426,E2 -22734.426} C_VEL
LIN {X 0,Y 198.237,Z 510.728,A -85,B 0,C 180,E1 -22736.667,E2 -22736.667} C_VEL
LIN {X 0,Y 197.117,Z 514.129,A -85,B 0,C 180,E1 -22737.669,E2 -22737.669} C_VEL
LIN {X 0,Y 192.459,Z 523.022,A -85,B 0,C 180,E1 -22740.464,E2 -22740.464} C_VEL
LIN {X 0,Y 188.128,Z 530.822,A -85,B 0,C 180,E1 -22743.713,E2 -22743.713} C_VEL
LIN {X 0,Y 185.042,Z 535.976,A -85,B 0,C 180,E1 -22746.497,E2 -22746.497} C_VEL
LIN {X 0,Y 182.09,Z 540.549,A -85,B 0,C 180,E1 -22749.674,E2 -22749.674} C_VEL
LIN {X 0,Y 179.65,Z 544.051,A -85,B 0,C 180,E1 -22752.938,E2 -22752.938} C_VEL
LIN {X 0,Y 177.94,Z 546.577,A -85,B 0,C 180,E1 -22756.292,E2 -22756.292} C_VEL
LIN {X 0,Y 177.095,Z 547.775,A -85,B 0,C 180,E1 -22758.555,E2 -22758.555} C_VEL
LIN {X 0,Y 176.146,Z 548.934,A -85,B 0,C 180,E1 -22763.125,E2 -22763.125} C_VEL
LIN {X 0,Y 175.992,Z 548.775,A -85,B 0,C 180,E1 -22766.708,E2 -22766.708} C_VEL
LIN {X 0,Y 176.126,Z 547.786,A -85,B 0,C 180,E1 -22770,E2 -22770} C_VEL
LIN {X 0,Y 175.997,Z 545.904,A -85,B 0,C 180,E1 -22773.319,E2 -22773.319} C_VEL
LIN {X 0,Y 176.155,Z 542.863,A -85,B 0,C 180,E1 -22776.874,E2 -22776.874} C_VEL
LIN {X 0,Y 176.681,Z 538.837,A -85,B 0,C 180,E1 -22780.311,E2 -22780.311} C_VEL
LIN {X 0,Y 177.793,Z 532.605,A -85,B 0,C 180,E1 -22784.303,E2 -22784.303} C_VEL
LIN {X 0,Y 178.116,Z 531.203,A -85,B 0,C 180,E1 -22785.071,E2 -22785.071} C_VEL
LIN {X 0,Y 178.197,Z 528.061,A -85,B 0,C 180,E1 -22786.686,E2 -22786.686} C_VEL
LIN {X 0,Y 176.682,Z 522.522,A -85,B 0,C 180,E1 -22789.313,E2 -22789.313} C_VEL
LIN {X 0,Y 175.438,Z 516.382,A -85,B 0,C 180,E1 -22791.83,E2 -22791.83} C_VEL
LIN {X 0,Y 175.923,Z 512.295,A -85,B 0,C 180,E1 -22793.218,E2 -22793.218} C_VEL
LIN {X 0,Y 178.506,Z 502.419,A -85,B 0,C 180,E1 -22795.976,E2 -22795.976} C_VEL
LIN {X 0,Y 179.135,Z 498.982,A -85,B 0,C 180,E1 -22796.818,E2 -22796.818} C_VEL
LIN {X 0,Y 179.232,Z 487.726,A -85,B 0,C 180,E1 -22799.417,E2 -22799.417} C_VEL
LIN {X 0,Y 178.784,Z 476.104,A -85,B 0,C 180,E1 -22801.649,E2 -22801.649} C_VEL
LIN {X 0,Y 177.466,Z 464.772,A -85,B 0,C 180,E1 -22803.516,E2 -22803.516} C_VEL
LIN {X 0,Y 174.974,Z 451.565,A -85,B 0,C 180,E1 -22805.382,E2 -22805.382} C_VEL
LIN {X 0,Y 172.678,Z 442.496,A -85,B 0,C 180,E1 -22806.533,E2 -22806.533} C_VEL
LIN {X 0,Y 172.648,Z 440.427,A -85,B 0,C 180,E1 -22809.336,E2 -22809.336} C_VEL
LIN {X 0,Y 172.08,Z 437.226,A -85,B 0,C 180,E1 -22813.97,E2 -22813.97} C_VEL
LIN {X 0,Y 171.405,Z 434.139,A -85,B 0,C 180,E1 -22819.001,E2 -22819.001} C_VEL
LIN {X 0,Y 171.389,Z 434.139,A -85,B 0,C 180,E1 -22822.041,E2 -22822.041} C_VEL
LIN {X 0,Y 171.396,Z 434.137,A -85,B 0,C 180,E1 -22825.091,E2 -22825.091} C_VEL
LIN {X 0,Y 171.446,Z 434.115,A -85,B 0,C 180,E1 -22830.533,E2 -22830.533} C_VEL
LIN {X 0,Y 171.455,Z 434.124,A -85,B 0,C 180,E1 -22835.801,E2 -22835.801} C_VEL
LIN {X 0,Y 171.575,Z 434.098,A -85,B 0,C 180,E1 -22840.871,E2 -22840.871} C_VEL
LIN {X 0,Y 171.57,Z 434.097,A -85,B 0,C 180,E1 -22845.772,E2 -22845.772} C_VEL
LIN {X 0,Y 171.899,Z 434.072,A -85,B 0,C 180,E1 -22850.587,E2 -22850.587} C_VEL
LIN {X 0,Y 171.819,Z 434.053,A -85,B 0,C 180,E1 -22855.307,E2 -22855.307} C_VEL
LIN {X 0,Y 172.33,Z 434.003,A -85,B 0,C 180,E1 -22860,E2 -22860} C_VEL
LIN {X 0,Y 171.82,Z 434.081,A -85,B 0,C 180,E1 -22864.692,E2 -22864.692} C_VEL
LIN {X 0,Y 171.886,Z 434.046,A -85,B 0,C 180,E1 -22869.413,E2 -22869.413} C_VEL
LIN {X 0,Y 171.573,Z 434.094,A -85,B 0,C 180,E1 -22874.227,E2 -22874.227} C_VEL
LIN {X 0,Y 171.54,Z 434.117,A -85,B 0,C 180,E1 -22879.562,E2 -22879.562} C_VEL
LIN {X 0,Y 171.458,Z 434.128,A -85,B 0,C 180,E1 -22885.611,E2 -22885.611} C_VEL
LIN {X 0,Y 171.436,Z 434.127,A -85,B 0,C 180,E1 -22890.586,E2 -22890.586} C_VEL
LIN {X 0,Y 171.403,Z 434.127,A -85,B 0,C 180,E1 -22895.032,E2 -22895.032} C_VEL
LIN {X 0,Y 171.435,Z 434.129,A -85,B 0,C 180,E1 -22898.842,E2 -22898.842} C_VEL
LIN {X 0,Y 171.45,Z 434.128,A -85,B 0,C 180,E1 -22904.175,E2 -22904.175} C_VEL
LIN {X 0,Y 171.433,Z 434.129,A -85,B 0,C 180,E1 -22909.011,E2 -22909.011} C_VEL
LIN {X 0,Y 171.44,Z 434.129,A -85,B 0,C 180,E1 -22912.056,E2 -22912.056} C_VEL
LIN {X 0,Y 171.418,Z 434.133,A -85,B 0,C 180,E1 -22917.794,E2 -22917.794} C_VEL
LIN {X 0,Y 171.448,Z 434.129,A -85,B 0,C 180,E1 -22920.535,E2 -22920.535} C_VEL
LIN {X 0,Y 171.587,Z 434.129,A -85,B 0,C 180,E1 -22926.464,E2 -22926.464} C_VEL
LIN {X 0,Y 171.643,Z 434.756,A -85,B 0,C 180,E1 -22927.401,E2 -22927.401} C_VEL
LIN {X 0,Y 172.71,Z 437.858,A -85,B 0,C 180,E1 -22927.839,E2 -22927.839} C_VEL
LIN {X 0,Y 176.746,Z 450.434,A -85,B 0,C 180,E1 -22929.774,E2 -22929.774} C_VEL
LIN {X 0,Y 179.254,Z 462.039,A -85,B 0,C 180,E1 -22931.721,E2 -22931.721} C_VEL
LIN {X 0,Y 180.879,Z 473.093,A -85,B 0,C 180,E1 -22933.846,E2 -22933.846} C_VEL
LIN {X 0,Y 181.495,Z 482.538,A -85,B 0,C 180,E1 -22935.886,E2 -22935.886} C_VEL
LIN {X 0,Y 179.342,Z 492.533,A -85,B 0,C 180,E1 -22938.112,E2 -22938.112} C_VEL
LIN {X 0,Y 176.779,Z 502.409,A -85,B 0,C 180,E1 -22940.85,E2 -22940.85} C_VEL
LIN {X 0,Y 174.55,Z 510.46,A -85,B 0,C 180,E1 -22943.643,E2 -22943.643} C_VEL
LIN {X 0,Y 172.388,Z 518.345,A -85,B 0,C 180,E1 -22947.079,E2 -22947.079} C_VEL
LIN {X 0,Y 171.136,Z 523.683,A -85,B 0,C 180,E1 -22950,E2 -22950} C_VEL
LIN {X 0,Y 170.01,Z 528.896,A -85,B 0,C 180,E1 -22953.555,E2 -22953.555} C_VEL
LIN {X 0,Y 169.219,Z 532.957,A -85,B 0,C 180,E1 -22957.158,E2 -22957.158} C_VEL
LIN {X 0,Y 168.798,Z 535.059,A -85,B 0,C 180,E1 -22959.587,E2 -22959.587} C_VEL
LIN {X 0,Y 168.579,Z 536.734,A -85,B 0,C 180,E1 -22962.032,E2 -22962.032} C_VEL
LIN {X 0,Y 168.579,Z 537.997,A -85,B 0,C 180,E1 -22964.486,E2 -22964.486} C_VEL
LIN {X 0,Y 168.737,Z 538.808,A -85,B 0,C 180,E1 -22966.951,E2 -22966.951} C_VEL
LIN {X 0,Y 169.081,Z 539.203,A -85,B 0,C 180,E1 -22969.422,E2 -22969.422} C_VEL
LIN {X 0,Y 169.599,Z 539.198,A -85,B 0,C 180,E1 -22971.898,E2 -22971.898} C_VEL
LIN {X 0,Y 170.63,Z 538.563,A -85,B 0,C 180,E1 -22975.022,E2 -22975.022} C_VEL
LIN {X 0,Y 172.605,Z 536.585,A -85,B 0,C 180,E1 -22979.249,E2 -22979.249} C_VEL
LIN {X 0,Y 174.591,Z 534.266,A -85,B 0,C 180,E1 -22982.293,E2 -22982.293} C_VEL
LIN {X 0,Y 177.984,Z 529.845,A -85,B 0,C 180,E1 -22986.32,E2 -22986.32} C_VEL
LIN {X 0,Y 181.63,Z 524.634,A -85,B 0,C 180,E1 -22989.729,E2 -22989.729} C_VEL
LIN {X 0,Y 185.763,Z 518.145,A -85,B 0,C 180,E1 -22992.921,E2 -22992.921} C_VEL
LIN {X 0,Y 190.315,Z 510.16,A -85,B 0,C 180,E1 -22995.91,E2 -22995.91} C_VEL
LIN {X 0,Y 194.807,Z 501.322,A -85,B 0,C 180,E1 -22998.468,E2 -22998.468} C_VEL
LIN {X 0,Y 195.258,Z 493.98,A -85,B 0,C 180,E1 -23000.959,E2 -23000.959} C_VEL
LIN {X 0,Y 194.737,Z 485.572,A -85,B 0,C 180,E1 -23003.752,E2 -23003.752} C_VEL
LIN {X 0,Y 193.427,Z 477.599,A -85,B 0,C 180,E1 -23006.415,E2 -23006.415} C_VEL
LIN {X 0,Y 190.725,Z 468.961,A -85,B 0,C 180,E1 -23009.558,E2 -23009.558} C_VEL
LIN {X 0,Y 187.485,Z 461.666,A -85,B 0,C 180,E1 -23012.522,E2 -23012.522} C_VEL
LIN {X 0,Y 184.94,Z 456.857,A -85,B 0,C 180,E1 -23014.69,E2 -23014.69} C_VEL
LIN {X 0,Y 183.214,Z 453.357,A -85,B 0,C 180,E1 -23016.249,E2 -23016.249} C_VEL
LIN {X 0,Y 180.828,Z 449.837,A -85,B 0,C 180,E1 -23018.183,E2 -23018.183} C_VEL
LIN {X 0,Y 180.002,Z 448.194,A -85,B 0,C 180,E1 -23018.979,E2 -23018.979} C_VEL
LIN {X 0,Y 177.618,Z 445.379,A -85,B 0,C 180,E1 -23020.948,E2 -23020.948} C_VEL
LIN {X 0,Y 176.484,Z 442.8,A -85,B 0,C 180,E1 -23022.174,E2 -23022.174} C_VEL
LIN {X 0,Y 173.729,Z 440.32,A -85,B 0,C 180,E1 -23024.605,E2 -23024.605} C_VEL
LIN {X 0,Y 172.343,Z 437.594,A -85,B 0,C 180,E1 -23026.214,E2 -23026.214} C_VEL
LIN {X 0,Y 172.142,Z 436.849,A -85,B 0,C 180,E1 -23026.574,E2 -23026.574} C_VEL
LIN {X 0,Y 172.248,Z 436.161,A -85,B 0,C 180,E1 -23030.607,E2 -23030.607} C_VEL
LIN {X 0,Y 172.122,Z 435.69,A -85,B 0,C 180,E1 -23035.316,E2 -23035.316} C_VEL
LIN {X 0,Y 172.559,Z 435.35,A -85,B 0,C 180,E1 -23040,E2 -23040} C_VEL
LIN {X 0,Y 172.196,Z 435.677,A -85,B 0,C 180,E1 -23047.033,E2 -23047.033} C_VEL
LIN {X 0,Y 172.129,Z 436.204,A -85,B 0,C 180,E1 -23051.506,E2 -23051.506} C_VEL
LIN {X 0,Y 172.111,Z 437.101,A -85,B 0,C 180,E1 -23056.609,E2 -23056.609} C_VEL
LIN {X 0,Y 172.211,Z 437.911,A -85,B 0,C 180,E1 -23060.178,E2 -23060.178} C_VEL
LIN {X 0,Y 172.357,Z 439.025,A -85,B 0,C 180,E1 -23064.065,E2 -23064.065} C_VEL
LIN {X 0,Y 172.572,Z 440.377,A -85,B 0,C 180,E1 -23067.927,E2 -23067.927} C_VEL
LIN {X 0,Y 173.595,Z 443.118,A -85,B 0,C 180,E1 -23069.174,E2 -23069.174} C_VEL
LIN {X 0,Y 176.366,Z 446.451,A -85,B 0,C 180,E1 -23071.703,E2 -23071.703} C_VEL
LIN {X 0,Y 177.17,Z 447.377,A -85,B 0,C 180,E1 -23072.38,E2 -23072.38} C_VEL
LIN {X 0,Y 179.03,Z 451.22,A -85,B 0,C 180,E1 -23074.195,E2 -23074.195} C_VEL
LIN {X 0,Y 180.957,Z 453.71,A -85,B 0,C 180,E1 -23075.714,E2 -23075.714} C_VEL
LIN {X 0,Y 182.866,Z 457.552,A -85,B 0,C 180,E1 -23077.401,E2 -23077.401} C_VEL
LIN {X 0,Y 184.649,Z 460.969,A -85,B 0,C 180,E1 -23078.904,E2 -23078.904} C_VEL
LIN {X 0,Y 187.727,Z 467.339,A -85,B 0,C 180,E1 -23081.519,E2 -23081.519} C_VEL
LIN {X 0,Y 190.854,Z 475.147,A -85,B 0,C 180,E1 -23084.4,E2 -23084.4} C_VEL
LIN {X 0,Y 192.8,Z 482.452,A -85,B 0,C 180,E1 -23086.807,E2 -23086.807} C_VEL
LIN {X 0,Y 193.568,Z 490.725,A -85,B 0,C 180,E1 -23089.192,E2 -23089.192} C_VEL
LIN {X 0,Y 193.487,Z 499.904,A -85,B 0,C 180,E1 -23091.867,E2 -23091.867} C_VEL
LIN {X 0,Y 192.796,Z 507.737,A -85,B 0,C 180,E1 -23094.321,E2 -23094.321} C_VEL
LIN {X 0,Y 191.789,Z 512.976,A -85,B 0,C 180,E1 -23096.025,E2 -23096.025} C_VEL
LIN {X 0,Y 188.668,Z 519.205,A -85,B 0,C 180,E1 -23097.939,E2 -23097.939} C_VEL
LIN {X 0,Y 184.149,Z 527.089,A -85,B 0,C 180,E1 -23100.883,E2 -23100.883} C_VEL
LIN {X 0,Y 180.963,Z 532.458,A -85,B 0,C 180,E1 -23103.486,E2 -23103.486} C_VEL
LIN {X 0,Y 177.422,Z 537.714,A -85,B 0,C 180,E1 -23106.664,E2 -23106.664} C_VEL
LIN {X 0,Y 174.487,Z 541.846,A -85,B 0,C 180,E1 -23109.979,E2 -23109.979} C_VEL
LIN {X 0,Y 172.139,Z 544.951,A -85,B 0,C 180,E1 -23113.394,E2 -23113.394} C_VEL
LIN {X 0,Y 171.019,Z 546.515,A -85,B 0,C 180,E1 -23115.725,E2 -23115.725} C_VEL
LIN {X 0,Y 170.118,Z 547.653,A -85,B 0,C 180,E1 -23118.079,E2 -23118.079} C_VEL
LIN {X 0,Y 169.099,Z 548.745,A -85,B 0,C 180,E1 -23122.837,E2 -23122.837} C_VEL
LIN {X 0,Y 168.901,Z 548.438,A -85,B 0,C 180,E1 -23127.025,E2 -23127.025} C_VEL
LIN {X 0,Y 169.034,Z 547.471,A -85,B 0,C 180,E1 -23130,E2 -23130} C_VEL
LIN {X 0,Y 168.912,Z 545.815,A -85,B 0,C 180,E1 -23133.042,E2 -23133.042} C_VEL
LIN {X 0,Y 169.108,Z 542.422,A -85,B 0,C 180,E1 -23137.162,E2 -23137.162} C_VEL
LIN {X 0,Y 169.672,Z 538.321,A -85,B 0,C 180,E1 -23140.742,E2 -23140.742} C_VEL
LIN {X 0,Y 170.878,Z 531.999,A -85,B 0,C 180,E1 -23144.895,E2 -23144.895} C_VEL
LIN {X 0,Y 172.704,Z 525.117,A -85,B 0,C 180,E1 -23148.383,E2 -23148.383} C_VEL
LIN {X 0,Y 174.875,Z 516.949,A -85,B 0,C 180,E1 -23151.651,E2 -23151.651} C_VEL
LIN {X 0,Y 175.923,Z 512.295,A -85,B 0,C 180,E1 -23153.218,E2 -23153.218} C_VEL
LIN {X 0,Y 176.396,Z 508.086,A -85,B 0,C 180,E1 -23154.545,E2 -23154.545} C_VEL
LIN {X 0,Y 175.794,Z 503.816,A -85,B 0,C 180,E1 -23155.889,E2 -23155.889} C_VEL
LIN {X 0,Y 173.41,Z 495.074,A -85,B 0,C 180,E1 -23158.522,E2 -23158.522} C_VEL
LIN {X 0,Y 172.549,Z 488.695,A -85,B 0,C 180,E1 -23160.136,E2 -23160.136} C_VEL
LIN {X 0,Y 172.24,Z 477.576,A -85,B 0,C 180,E1 -23162.413,E2 -23162.413} C_VEL
LIN {X 0,Y 171.016,Z 466.024,A -85,B 0,C 180,E1 -23164.463,E2 -23164.463} C_VEL
LIN {X 0,Y 168.752,Z 453.295,A -85,B 0,C 180,E1 -23166.403,E2 -23166.403} C_VEL
LIN {X 0,Y 166.5,Z 445.203,A -85,B 0,C 180,E1 -23167.568,E2 -23167.568} C_VEL
LIN {X 0,Y 165.687,Z 442.284,A -85,B 0,C 180,E1 -23167.975,E2 -23167.975} C_VEL
LIN {X 0,Y 165.537,Z 440.775,A -85,B 0,C 180,E1 -23170.163,E2 -23170.163} C_VEL
LIN {X 0,Y 165.109,Z 438.476,A -85,B 0,C 180,E1 -23173.645,E2 -23173.645} C_VEL
LIN {X 0,Y 164.35,Z 435.018,A -85,B 0,C 180,E1 -23179.297,E2 -23179.297} C_VEL
LIN {X 0,Y 164.328,Z 435.017,A -85,B 0,C 180,E1 -23184.348,E2 -23184.348} C_VEL
LIN {X 0,Y 164.387,Z 435.004,A -85,B 0,C 180,E1 -23189.133,E2 -23189.133} C_VEL
LIN {X 0,Y 164.414,Z 434.994,A -85,B 0,C 180,E1 -23194.693,E2 -23194.693} C_VEL
LIN {X 0,Y 164.482,Z 434.987,A -85,B 0,C 180,E1 -23200.05,E2 -23200.05} C_VEL
LIN {X 0,Y 164.499,Z 434.968,A -85,B 0,C 180,E1 -23205.146,E2 -23205.146} C_VEL
LIN {X 0,Y 164.829,Z 434.953,A -85,B 0,C 180,E1 -23210.18,E2 -23210.18} C_VEL
LIN {X 0,Y 164.857,Z 434.94,A -85,B 0,C 180,E1 -23212.652,E2 -23212.652} C_VEL
LIN {X 0,Y 165.293,Z 434.879,A -85,B 0,C 180,E1 -23220,E2 -23220} C_VEL
LIN {X 0,Y 164.77,Z 434.959,A -85,B 0,C 180,E1 -23224.893,E2 -23224.893} C_VEL
LIN {X 0,Y 164.85,Z 434.94,A -85,B 0,C 180,E1 -23227.348,E2 -23227.348} C_VEL
LIN {X 0,Y 164.738,Z 434.924,A -85,B 0,C 180,E1 -23231.131,E2 -23231.131} C_VEL
LIN {X 0,Y 164.479,Z 434.995,A -85,B 0,C 180,E1 -23237.403,E2 -23237.403} C_VEL
LIN {X 0,Y 164.47,Z 434.995,A -85,B 0,C 180,E1 -23239.989,E2 -23239.989} C_VEL
LIN {X 0,Y 164.384,Z 435.008,A -85,B 0,C 180,E1 -23246.13,E2 -23246.13} C_VEL
LIN {X 0,Y 164.37,Z 435.008,A -85,B 0,C 180,E1 -23251.227,E2 -23251.227} C_VEL
LIN {X 0,Y 164.348,Z 435.008,A -85,B 0,C 180,E1 -23256.775,E2 -23256.775} C_VEL
LIN {X 0,Y 164.372,Z 435.008,A -85,B 0,C 180,E1 -23259.892,E2 -23259.892} C_VEL
LIN {X 0,Y 164.388,Z 435.007,A -85,B 0,C 180,E1 -23263.384,E2 -23263.384} C_VEL
LIN {X 0,Y 164.394,Z 435.005,A -85,B 0,C 180,E1 -23266.844,E2 -23266.844} C_VEL
LIN {X 0,Y 164.375,Z 435.009,A -85,B 0,C 180,E1 -23270.318,E2 -23270.318} C_VEL
LIN {X 0,Y 164.346,Z 435.011,A -85,B 0,C 180,E1 -23274.341,E2 -23274.341} C_VEL
LIN {X 0,Y 164.39,Z 435.008,A -85,B 0,C 180,E1 -23279.136,E2 -23279.136} C_VEL
LIN {X 0,Y 164.524,Z 434.994,A -85,B 0,C 180,E1 -23285.877,E2 -23285.877} C_VEL
LIN {X 0,Y 165.546,Z 437.837,A -85,B 0,C 180,E1 -23286.351,E2 -23286.351} C_VEL
LIN {X 0,Y 168.121,Z 444.542,A -85,B 0,C 180,E1 -23287.492,E2 -23287.492} C_VEL
LIN {X 0,Y 170.876,Z 453.974,A -85,B 0,C 180,E1 -23289.118,E2 -23289.118} C_VEL
LIN {X 0,Y 173.152,Z 465.651,A -85,B 0,C 180,E1 -23291.269,E2 -23291.269} C_VEL
LIN {X 0,Y 174.43,Z 475.877,A -85,B 0,C 180,E1 -23293.398,E2 -23293.398} C_VEL
LIN {X 0,Y 174.752,Z 484.237,A -85,B 0,C 180,E1 -23295.329,E2 -23295.329} C_VEL
LIN {X 0,Y 172.138,Z 494.851,A -85,B 0,C 180,E1 -23297.84,E2 -23297.84} C_VEL
LIN {X 0,Y 169.754,Z 503.672,A -85,B 0,C 180,E1 -23300.468,E2 -23300.468} C_VEL
LIN {X 0,Y 167.088,Z 512.909,A -85,B 0,C 180,E1 -23303.965,E2 -23303.965} C_VEL
LIN {X 0,Y 164.99,Z 520.335,A -85,B 0,C 180,E1 -23307.559,E2 -23307.559} C_VEL
LIN {X 0,Y 163.545,Z 526.281,A -85,B 0,C 180,E1 -23311.232,E2 -23311.232} C_VEL
LIN {X 0,Y 162.417,Z 531.656,A -85,B 0,C 180,E1 -23315.597,E2 -23315.597} C_VEL
LIN {X 0,Y 161.644,Z 535.538,A -85,B 0,C 180,E1 -23320.016,E2 -23320.016} C_VEL
LIN {X 0,Y 161.461,Z 537.163,A -85,B 0,C 180,E1 -23322.571,E2 -23322.571} C_VEL
LIN {X 0,Y 161.663,Z 538.943,A -85,B 0,C 180,E1 -23326.981,E2 -23326.981} C_VEL
LIN {X 0,Y 162.129,Z 539.439,A -85,B 0,C 180,E1 -23330.291,E2 -23330.291} C_VEL
LIN {X 0,Y 162.746,Z 539.384,A -85,B 0,C 180,E1 -23332.871,E2 -23332.871} C_VEL
LIN {X 0,Y 163.738,Z 538.795,A -85,B 0,C 180,E1 -23335.663,E2 -23335.663} C_VEL
LIN {X 0,Y 166.131,Z 536.574,A -85,B 0,C 180,E1 -23340.507,E2 -23340.507} C_VEL
LIN {X 0,Y 168.687,Z 533.764,A -85,B 0,C 180,E1 -23344.081,E2 -23344.081} C_VEL
LIN {X 0,Y 172.033,Z 529.624,A -85,B 0,C 180,E1 -23347.791,E2 -23347.791} C_VEL
LIN {X 0,Y 175.921,Z 524.346,A -85,B 0,C 180,E1 -23351.236,E2 -23351.236} C_VEL
LIN {X 0,Y 180.372,Z 517.608,A -85,B 0,C 180,E1 -23354.535,E2 -23354.535} C_VEL
LIN {X 0,Y 185.381,Z 509.16,A -85,B 0,C 180,E1 -23357.668,E2 -23357.668} C_VEL
LIN {X 0,Y 188.779,Z 502.609,A -85,B 0,C 180,E1 -23359.601,E2 -23359.601} C_VEL
LIN {X 0,Y 189.267,Z 495.705,A -85,B 0,C 180,E1 -23362.13,E2 -23362.13} C_VEL
LIN {X 0,Y 189.008,Z 487.963,A -85,B 0,C 180,E1 -23364.888,E2 -23364.888} C_VEL
LIN {X 0,Y 187.94,Z 480.712,A -85,B 0,C 180,E1 -23367.502,E2 -23367.502} C_VEL
LIN {X 0,Y 185.738,Z 473.057,A -85,B 0,C 180,E1 -23370.535,E2 -23370.535} C_VEL
LIN {X 0,Y 183.262,Z 466.892,A -85,B 0,C 180,E1 -23373.218,E2 -23373.218} C_VEL
LIN {X 0,Y 181.73,Z 463.409,A -85,B 0,C 180,E1 -23374.824,E2 -23374.824} C_VEL
LIN {X 0,Y 179.604,Z 459.043,A -85,B 0,C 180,E1 -23376.965,E2 -23376.965} C_VEL
LIN {X 0,Y 177.844,Z 456.411,A -85,B 0,C 180,E1 -23378.56,E2 -23378.56} C_VEL
LIN {X 0,Y 176.103,Z 453.492,A -85,B 0,C 180,E1 -23380.323,E2 -23380.323} C_VEL
LIN {X 0,Y 174.092,Z 450.01,A -85,B 0,C 180,E1 -23382.452,E2 -23382.452} C_VEL
LIN {X 0,Y 173.558,Z 448.982,A -85,B 0,C 180,E1 -23383.08,E2 -23383.08} C_VEL
LIN {X 0,Y 170.994,Z 446.124,A -85,B 0,C 180,E1 -23385.724,E2 -23385.724} C_VEL
LIN {X 0,Y 169.767,Z 443.391,A -85,B 0,C 180,E1 -23387.448,E2 -23387.448} C_VEL
LIN {X 0,Y 166.757,Z 440.645,A -85,B 0,C 180,E1 -23391.213,E2 -23391.213} C_VEL
LIN {X 0,Y 165.248,Z 437.518,A -85,B 0,C 180,E1 -23394.203,E2 -23394.203} C_VEL
LIN {X 0,Y 165.674,Z 437.096,A -85,B 0,C 180,E1 -23400,E2 -23400} C_VEL
LIN {X 0,Y 165.319,Z 437.465,A -85,B 0,C 180,E1 -23407.328,E2 -23407.328} C_VEL
LIN {X 0,Y 165.243,Z 438.037,A -85,B 0,C 180,E1 -23411.983,E2 -23411.983} C_VEL
LIN {X 0,Y 165.238,Z 438.975,A -85,B 0,C 180,E1 -23417.322,E2 -23417.322} C_VEL
LIN {X 0,Y 165.351,Z 439.706,A -85,B 0,C 180,E1 -23420.172,E2 -23420.172} C_VEL
LIN {X 0,Y 166.551,Z 442.817,A -85,B 0,C 180,E1 -23422.484,E2 -23422.484} C_VEL
LIN {X 0,Y 169.584,Z 446.248,A -85,B 0,C 180,E1 -23426.346,E2 -23426.346} C_VEL
LIN {X 0,Y 170.312,Z 447.053,A -85,B 0,C 180,E1 -23427.162,E2 -23427.162} C_VEL
LIN {X 0,Y 171.752,Z 450.392,A -85,B 0,C 180,E1 -23429.073,E2 -23429.073} C_VEL
LIN {X 0,Y 174.261,Z 453.418,A -85,B 0,C 180,E1 -23431.537,E2 -23431.537} C_VEL
LIN {X 0,Y 176.166,Z 457.492,A -85,B 0,C 180,E1 -23433.644,E2 -23433.644} C_VEL
LIN {X 0,Y 177.259,Z 458.896,A -85,B 0,C 180,E1 -23434.602,E2 -23434.602} C_VEL
LIN {X 0,Y 179.311,Z 463.288,A -85,B 0,C 180,E1 -23436.707,E2 -23436.707} C_VEL
LIN {X 0,Y 182.218,Z 469.396,A -85,B 0,C 180,E1 -23439.522,E2 -23439.522} C_VEL
LIN {X 0,Y 185.468,Z 477.931,A -85,B 0,C 180,E1 -23443.007,E2 -23443.007} C_VEL
LIN {X 0,Y 187.266,Z 484.794,A -85,B 0,C 180,E1 -23445.485,E2 -23445.485} C_VEL
LIN {X 0,Y 187.875,Z 493.309,A -85,B 0,C 180,E1 -23448.169,E2 -23448.169} C_VEL
LIN {X 0,Y 187.482,Z 502.412,A -85,B 0,C 180,E1 -23451.025,E2 -23451.025} C_VEL
LIN {X 0,Y 186.515,Z 510.086,A -85,B 0,C 180,E1 -23453.597,E2 -23453.597} C_VEL
